// TwinCAT 3 PLC project PLCProject
// ProgramVersion: 3.1.4024.0
// libraries:
//   Tc2_MC2, * (Beckhoff Automation GmbH)
//   Tc2_MC2_Drive, * (Beckhoff Automation GmbH)
//   Tc2_NC, * (Beckhoff Automation GmbH)
//   Tc2_Standard, * (Beckhoff Automation GmbH)
//   Tc2_System, * (Beckhoff Automation GmbH)
//   Tc2_Utilities, * (Beckhoff Automation GmbH)
//   Tc3_EventLogger, * (Beckhoff Automation GmbH)
//   Tc3_Module, * (Beckhoff Automation GmbH)
// project tree:
//   DUTs/Coil Shapes/ pancake_params_0.TcDUT, racetrack_params_1.TcDUT
//   DUTs/HMI Datagrids/Inputs/ general_input_datagrid_params.TcDUT, misc_settings_input_datagrid_params.TcDUT (not stored), payoff_input_datagrid_params.TcDUT, pickup_input_datagrid_params.TcDUT
//   DUTs/HMI Datagrids/Outputs/ motor_info_datagrid.TcDUT, motor_state_datagrid.TcDUT (not stored), output_error_datagrid.TcDUT, overview_outputs_datagrid.TcDUT (not stored), payoff_output_datagrid_params.TcDUT, pickup_output_datagrid_params.TcDUT (not stored), turncount_output_datagrid.TcDUT
//   DUTs/Input Bounds/ input_bounds.TcDUT
//   DUTs/ tape_info.TcDUT
//   GVLs/ GVL.TcGVL
//   / PlcTask.TcTTO, RecipeManager.TcRMO (not stored)
//   POUs/ FB_Axis.TcPOU, FB_EventLogger.TcPOU, FB_fileReadWrite.TcPOU, FB_hmi_connection.TcPOU, FB_WindingControl.TcPOU, MAIN.TcPOU
// real-time tasks:
//   TASK PlcTask: cycle T#10ms, priority 20, ADS port 350
// motion (NC):
//   TASK NC-Task 1 SAF: cycle T#2ms, priority 4, ADS port 501
//   TASK NC-Task 1 SVB: cycle T#10ms, priority 8, ADS port 511
//   AXIS Pickup (id 1)
//     General: UnitName=°
//     Dynamic: Acceleration=2990.4, Deceleration=2990.4, Jerk=8971.19
//     Velo: RefSearch=19.93598, RefSync=19.93598, SlowManual=99.6799, FastManual=598.0794, Fast=1993.598, Maximum=1993.598
//     OtherSettings: AllowMotionCmdToSlave=true
//     encoder EncType=8
//       EncPara: ScaleFactorNumerator=360, ScaleFactorDenominator=10485760, MaxCount=#xffffffff
//     drive DrvType=9
//       DrvPara: MaxCount=#xffffffff, DriveControlDWord=#x00030100
//         Analog: VeloReferenz=2192.9578, VeloScale=1.02400649589962, TorqueSetpointScale=10, ScaleFactorActTorque=0.1
//         TimeComp: TaskDelayCycles=1
//     controller CtrType=1
//       CtrPara: PriorControlFactor=1
//         Observer: BandWidth=20
//   AXIS Payoff 1 (id 2)
//     General: UnitName=°
//     Dynamic: Acceleration=805.38, Deceleration=805.38, Jerk=2416.14
//     Velo: RefSearch=5.3692, RefSync=5.3692, SlowManual=26.846, FastManual=161.076, Fast=536.92, Maximum=536.92
//     OtherSettings: AllowMotionCmdToSlave=true
//     encoder EncType=19
//       EncPara: ScaleFactorNumerator=360, ScaleFactorDenominator=62914560, MaxCount=#xffffffff
//     drive DrvType=16
//       DrvPara: MaxCount=#xffffffff, DriveControlDWord=#x00020100
//         Analog: VeloReferenz=590.612, VeloScale=32, TorqueSetpointScale=10, ScaleFactorActTorque=0.1
//         TimeComp: TaskDelayCycles=1
//     controller CtrType=1
//       CtrPara: PriorControlFactor=1
//         Observer: BandWidth=20
//   AXIS Payoff 2 (id 3)
//     General: UnitName=°
//     Dynamic: Acceleration=805.38, Deceleration=805.38, Jerk=2416.14
//     Velo: RefSearch=5.3692, RefSync=5.3692, SlowManual=26.846, FastManual=161.076, Fast=536.92, Maximum=536.92
//     OtherSettings: AllowMotionCmdToSlave=true
//     encoder EncType=19
//       EncPara: ScaleFactorNumerator=360, ScaleFactorDenominator=62914560, MaxCount=#xffffffff
//     drive DrvType=16
//       DrvPara: MaxCount=#xffffffff, DriveControlDWord=#x00020100
//         Analog: VeloReferenz=590.612, VeloScale=32, TorqueSetpointScale=10, ScaleFactorActTorque=0.1
//         TimeComp: TaskDelayCycles=1
//     controller CtrType=1
//       CtrPara: PriorControlFactor=1
//         Observer: BandWidth=20
//   AXIS Payoff 3 (id 4)
//     General: UnitName=°
//     Dynamic: Acceleration=805.38, Deceleration=805.38, Jerk=2416.14
//     Velo: RefSearch=5.3692, RefSync=5.3692, SlowManual=26.846, FastManual=161.076, Fast=536.92, Maximum=536.92
//     OtherSettings: AllowMotionCmdToSlave=true
//     encoder EncType=19
//       EncPara: ScaleFactorNumerator=360, ScaleFactorDenominator=62914560, MaxCount=#xffffffff
//     drive DrvType=16
//       DrvPara: MaxCount=#xffffffff, DriveControlDWord=#x00020100
//         Analog: VeloReferenz=590.612, VeloScale=32, TorqueSetpointScale=10, ScaleFactorActTorque=0.1
//         TimeComp: TaskDelayCycles=1
//     controller CtrType=1
//       CtrPara: PriorControlFactor=1
//         Observer: BandWidth=20
// I/O:
//   DEVICE Device 1 (EtherCAT), AmsNetId 5.143.168.64.2.1
//     Term 9 (EK1200) [EK1200-5000 EtherCAT Power supply (2A E-Bus)]
//       Term 2 (EL3002) [EL3002 2Ch. Ana. Input +/-10V]
//       Term 3 (EL1859) [EL1859 8Ch. Dig. Input 24V, 3ms, 8Ch. Dig. Output 24V, 0.5A]
//       Term 4 (EL6070-0033) [EL6070-0033 1Ch. Licence key terminal, individual licences]
//       Term 11 (ELM7222-0011) [ELM7222-0011 2Ch. Servo Terminal (DS402, 48 V, 8 A RMS, OCT)]
//         startup 8195:21 := 0E01 // Motor Settings Ch.1 / Commutation offset
//         startup 24704:0 := 10270000 // Max motor speed Ch.1
//         startup 8196:19 := 0000 // Brake Settings Ch.1 / Emergency application timeout
//         startup 8194:51 := 0A00 // Amplifier Settings Ch.1 / Stand still window
//         startup 8194:19 := 7600 // Amplifier Settings Ch.1 / Current loop proportional gain
//         startup 8194:18 := 1300 // Amplifier Settings Ch.1 / Current loop integral time
//         startup 8194:21 := 24010000 // Amplifier Settings Ch.1 / Velocity loop proportional gain
//         startup 8194:20 := 96000000 // Amplifier Settings Ch.1 / Velocity loop integral time
//       Term 12 (ELM7222-0011) [ELM7222-0011 2Ch. Servo Terminal (DS402, 48 V, 8 A RMS, OCT)]
//         startup 8195:21 := 0E01 // Motor Settings Ch.1 / Commutation offset
//         startup 24704:0 := 10270000 // Max motor speed Ch.1
//         startup 8196:19 := 0000 // Brake Settings Ch.1 / Emergency application timeout
//         startup 8194:51 := 0A00 // Amplifier Settings Ch.1 / Stand still window
//         startup 8194:19 := 7600 // Amplifier Settings Ch.1 / Current loop proportional gain
//         startup 8194:18 := 1300 // Amplifier Settings Ch.1 / Current loop integral time
//         startup 8194:21 := 24010000 // Amplifier Settings Ch.1 / Velocity loop proportional gain
//         startup 8194:20 := 96000000 // Amplifier Settings Ch.1 / Velocity loop integral time
//         startup 10243:21 := 0E01 // Motor Settings Ch.2 / Commutation offset
//         startup 26752:0 := 10270000 // Max motor speed Ch.2
//         startup 10244:19 := 0000 // Brake Settings Ch.2 / Emergency application timeout
//         startup 10242:51 := 0A00 // Amplifier Settings Ch.2 / Stand still window
//         startup 10242:19 := 7600 // Amplifier Settings Ch.2 / Current loop proportional gain
//         startup 10242:18 := 1300 // Amplifier Settings Ch.2 / Current loop integral time
//         startup 10242:21 := 24010000 // Amplifier Settings Ch.2 / Velocity loop proportional gain
//         startup 10242:20 := 96000000 // Amplifier Settings Ch.2 / Velocity loop integral time
//       Term 13 (EK1110) [EK1110 EtherCAT extension]
//     Drive 16 (AX5103-0000-0214) [AX5103-0000-0214 EtherCAT Drive (SoE, 1 Ch.)]
// variable links:
//   NC-Task 1 SAF/Axes/Payoff 1 <-> Device 1 (EtherCAT)/Term 9 (EK1200)/Term 12 (ELM7222-0011)
//     Drive/Inputs/In/nDataIn1 <-> DS402 Following error actual value Channel 2/Following error actual value
//     Drive/Inputs/In/nDataIn3[0] <-> DS402 Torque actual value Channel 2/Torque actual value
//     Drive/Inputs/In/nDcOutputTime <-> InfoData/DcOutputShift
//     Drive/Inputs/In/nState1 <-> DS402 Statusword Channel 2/Statusword
//     Drive/Inputs/In/nState2 <-> DS402 Statusword Channel 2/Statusword @bit 8
//     Drive/Inputs/In/nState4 @bit 1 <-> WcState/InputToggle
//     Drive/Inputs/In/nState4 <-> WcState/WcState
//     Drive/Inputs/In/nState5 <-> DS402 Modes of operation display Channel 2/Modes of operation display
//     Drive/Outputs/Out/nCtrl1 <-> DS402 Controlword Channel 2/Controlword
//     Drive/Outputs/Out/nCtrl2 <-> DS402 Controlword Channel 2/Controlword @bit 8
//     Drive/Outputs/Out/nCtrl5 <-> DS402 Modes of operation Channel 2/Modes of operation
//     Drive/Outputs/Out/nDataOut1 <-> DS402 Target position Channel 2/Target position
//     Drive/Outputs/Out/nDataOut4[0] <-> DS402 Target torque Channel 2/Target torque
//     Drive/Outputs/Out/nDataOut5 <-> DS402 High velocity limit value Channel 2/High velocity limit value
//     Drive/Outputs/Out/nDataOut6 <-> DS402 Low velocity limit value Channel 2/Low velocity limit value
//     Enc/Inputs/In/nDataIn1 <-> DS402 Position actual value Channel 2/Position actual value
//     Enc/Inputs/In/nDcInputTime <-> InfoData/DcInputShift
//     Enc/Inputs/In/nState4 @bit 1 <-> WcState/InputToggle
//     Enc/Inputs/In/nState4 <-> WcState/WcState
//   NC-Task 1 SAF/Axes/Payoff 2 <-> Device 1 (EtherCAT)/Term 9 (EK1200)/Term 11 (ELM7222-0011)
//     Drive/Inputs/In/nDataIn1 <-> DS402 Following error actual value Channel 1/Following error actual value
//     Drive/Inputs/In/nDataIn3[0] <-> DS402 Torque actual value Channel 1/Torque actual value
//     Drive/Inputs/In/nDcOutputTime <-> InfoData/DcOutputShift
//     Drive/Inputs/In/nState1 <-> DS402 Statusword Channel 1/Statusword
//     Drive/Inputs/In/nState2 <-> DS402 Statusword Channel 1/Statusword @bit 8
//     Drive/Inputs/In/nState4 @bit 1 <-> WcState/InputToggle
//     Drive/Inputs/In/nState4 <-> WcState/WcState
//     Drive/Inputs/In/nState5 <-> DS402 Modes of operation display Channel 1/Modes of operation display
//     Drive/Outputs/Out/nCtrl1 <-> DS402 Controlword Channel 1/Controlword
//     Drive/Outputs/Out/nCtrl2 <-> DS402 Controlword Channel 1/Controlword @bit 8
//     Drive/Outputs/Out/nCtrl5 <-> DS402 Modes of operation Channel 1/Modes of operation
//     Drive/Outputs/Out/nDataOut1 <-> DS402 Target position Channel 1/Target position
//     Drive/Outputs/Out/nDataOut4[0] <-> DS402 Target torque Channel 1/Target torque
//     Drive/Outputs/Out/nDataOut5 <-> DS402 High velocity limit value Channel 1/High velocity limit value
//     Drive/Outputs/Out/nDataOut6 <-> DS402 Low velocity limit value Channel 1/Low velocity limit value
//     Enc/Inputs/In/nDataIn1 <-> DS402 Position actual value Channel 1/Position actual value
//     Enc/Inputs/In/nDcInputTime <-> InfoData/DcInputShift
//     Enc/Inputs/In/nState4 @bit 1 <-> WcState/InputToggle
//     Enc/Inputs/In/nState4 <-> WcState/WcState
//   NC-Task 1 SAF/Axes/Payoff 3 <-> Device 1 (EtherCAT)/Term 9 (EK1200)/Term 12 (ELM7222-0011)
//     Drive/Inputs/In/nDataIn1 <-> DS402 Following error actual value Channel 1/Following error actual value
//     Drive/Inputs/In/nDataIn3[0] <-> DS402 Torque actual value Channel 1/Torque actual value
//     Drive/Inputs/In/nDcOutputTime <-> InfoData/DcOutputShift
//     Drive/Inputs/In/nState1 <-> DS402 Statusword Channel 1/Statusword
//     Drive/Inputs/In/nState2 <-> DS402 Statusword Channel 1/Statusword @bit 8
//     Drive/Inputs/In/nState4 @bit 1 <-> WcState/InputToggle
//     Drive/Inputs/In/nState4 <-> WcState/WcState
//     Drive/Inputs/In/nState5 <-> DS402 Modes of operation display Channel 1/Modes of operation display
//     Drive/Outputs/Out/nCtrl1 <-> DS402 Controlword Channel 1/Controlword
//     Drive/Outputs/Out/nCtrl2 <-> DS402 Controlword Channel 1/Controlword @bit 8
//     Drive/Outputs/Out/nCtrl5 <-> DS402 Modes of operation Channel 1/Modes of operation
//     Drive/Outputs/Out/nDataOut1 <-> DS402 Target position Channel 1/Target position
//     Drive/Outputs/Out/nDataOut4[0] <-> DS402 Target torque Channel 1/Target torque
//     Drive/Outputs/Out/nDataOut5 <-> DS402 High velocity limit value Channel 1/High velocity limit value
//     Drive/Outputs/Out/nDataOut6 <-> DS402 Low velocity limit value Channel 1/Low velocity limit value
//     Enc/Inputs/In/nDataIn1 <-> DS402 Position actual value Channel 1/Position actual value
//     Enc/Inputs/In/nDcInputTime <-> InfoData/DcInputShift
//     Enc/Inputs/In/nState4 @bit 1 <-> WcState/InputToggle
//     Enc/Inputs/In/nState4 <-> WcState/WcState
//   NC-Task 1 SAF/Axes/Pickup <-> Device 1 (EtherCAT)/Drive 16 (AX5103-0000-0214)
//     Drive/Inputs/In/nDataIn1 <-> AT/Following distance
//     Drive/Inputs/In/nDataIn3[0] <-> AT/Torque/force feedback value
//     Drive/Inputs/In/nDcOutputTime <-> InfoData/DcOutputShift
//     Drive/Inputs/In/nState1 <-> AT/Drive status word @bit 8
//     Drive/Inputs/In/nState2 <-> AT/Drive status word
//     Drive/Inputs/In/nState4 @bit 1 <-> WcState/InputToggle
//     Drive/Inputs/In/nState4 <-> WcState/WcState
//     Drive/Outputs/Out/nCtrl1 <-> MDT/Master control word @bit 8
//     Drive/Outputs/Out/nDataOut1 <-> MDT/Position command value
//     Drive/Outputs/Out/nDataOut4[0] <-> MDT/Torque/force command value
//     Drive/Outputs/Out/nDataOut5 <-> MDT/High velocity limit value
//     Drive/Outputs/Out/nDataOut6 <-> MDT/Low velocity limit value
//     Enc/Inputs/In/nDataIn1 <-> AT/Position feedback 1 value
//     Enc/Inputs/In/nDcInputTime <-> InfoData/DcInputShift
//     Enc/Inputs/In/nState4 @bit 1 <-> WcState/InputToggle
//     Enc/Inputs/In/nState4 <-> WcState/WcState
//   PLCProject/PLCProject Instance <-> NC-Task 1 SAF/Axes/Payoff 1
//     PlcTask Inputs/MAIN.FB_WindingControl.payoff_axis_list[1].AXIS.NcToPlc <-> Outputs/ToPlc
//     PlcTask Outputs/MAIN.FB_WindingControl.payoff_axis_list[1].AXIS.PlcToNc <-> Inputs/FromPlc
//   PLCProject/PLCProject Instance <-> NC-Task 1 SAF/Axes/Payoff 2
//     PlcTask Inputs/MAIN.FB_WindingControl.payoff_axis_list[2].AXIS.NcToPlc <-> Outputs/ToPlc
//     PlcTask Outputs/MAIN.FB_WindingControl.payoff_axis_list[2].AXIS.PlcToNc <-> Inputs/FromPlc
//   PLCProject/PLCProject Instance <-> NC-Task 1 SAF/Axes/Payoff 3
//     PlcTask Inputs/MAIN.FB_WindingControl.payoff_axis_list[3].AXIS.NcToPlc <-> Outputs/ToPlc
//     PlcTask Outputs/MAIN.FB_WindingControl.payoff_axis_list[3].AXIS.PlcToNc <-> Inputs/FromPlc
//   PLCProject/PLCProject Instance <-> NC-Task 1 SAF/Axes/Pickup
//     PlcTask Inputs/MAIN.FB_WindingControl.pickup_axis_list[1].AXIS.NcToPlc <-> Outputs/ToPlc
//     PlcTask Outputs/MAIN.FB_WindingControl.pickup_axis_list[1].AXIS.PlcToNc <-> Inputs/FromPlc

CONFIGURATION PLCProject
    RESOURCE PLC ON TwinCAT3
        TASK PlcTask(INTERVAL := T#10ms, PRIORITY := 20);
        PROGRAM MAIN WITH PlcTask : MAIN;
    END_RESOURCE
END_CONFIGURATION

// ---- DUTs/Coil Shapes/pancake_params_0.TcDUT
TYPE pancake_params_0 :
STRUCT
	radius : LREAL := 200; // radius of pancake coil in mm
END_STRUCT
END_TYPE

// ---- DUTs/Coil Shapes/racetrack_params_1.TcDUT
//Defining our dimensions for our racetrack coil
TYPE racetrack_params_1 :
STRUCT
	length : LREAL := 150; //mm
	radius : LREAL := 100; //mm
END_STRUCT
END_TYPE

// ---- DUTs/HMI Datagrids/Inputs/general_input_datagrid_params.TcDUT
TYPE general_input_datagrid_params :
STRUCT
	tension : LREAL :=10;
	linspeed : LREAL:=0.5;
	unwinding : BOOL;
END_STRUCT
END_TYPE

// ---- DUTs/HMI Datagrids/Inputs/payoff_input_datagrid_params.TcDUT
TYPE payoff_input_datagrid_params :
STRUCT
	motor_name : STRING;
	tape_type : INT :=1;
	coil_type : INT :=1;
	radius : LREAL :=150;
	enabled : BOOL ;
END_STRUCT
END_TYPE

// ---- DUTs/HMI Datagrids/Inputs/pickup_input_datagrid_params.TcDUT
TYPE pickup_input_datagrid_params :
STRUCT
	motor_name : STRING;
	turn_count: INT :=1;
	coil_shape: INT :=0;
END_STRUCT
END_TYPE

// ---- DUTs/HMI Datagrids/Outputs/motor_info_datagrid.TcDUT
TYPE motor_info_datagrid :
STRUCT
	speed : LREAL;
	torque : LREAL;
	errortype : UDINT;
	errorid : UDINT;
	currentRadius: LREAL;
END_STRUCT
END_TYPE

// ---- DUTs/HMI Datagrids/Outputs/output_error_datagrid.TcDUT
TYPE output_error_datagrid :
STRUCT
	errorStatus : BOOL;
	errorID : UDINT;
END_STRUCT
END_TYPE

// ---- DUTs/HMI Datagrids/Outputs/payoff_output_datagrid_params.TcDUT
TYPE payoff_output_datagrid_params :
STRUCT
	motor_name: STRING;
	rpm : LREAL;
	linear_speed : LREAL;
	turn_count : LREAL;
	enabled : BOOL ;
END_STRUCT
END_TYPE

// ---- DUTs/HMI Datagrids/Outputs/turncount_output_datagrid.TcDUT
TYPE turncount_output_datagrid :
STRUCT
	
	pickupTC1 : LREAL;
	payoffTC1 : LREAL;
	payoffTC2 : LREAL;
	payoffTC3 : LREAL;
END_STRUCT
END_TYPE

// ---- DUTs/Input Bounds/input_bounds.TcDUT
//defines bounds for all HMI inputs
TYPE input_bounds :
STRUCT
	
	linear_speed_low : LREAL := 0.01; //(m/s)
	linear_speed_high: LREAL := 1.0;  //(m/s)

	tension_low : LREAL := 5; //(N)
	tension_high : LREAL := 20; //(N)
	
	turn_count_pickup_low : INT := 1;
	turn_count_pickup_high : INT := 1000;
	
	radius_payoff_low : LREAL:=GVL.MIN_MOUNT_RADIUS; //(mm)
	radius_payoff_high : LREAL:=GVL.MAX_PAYOFF_RADIUS-10; //(mm)
	
	radius_pickup_pancake_low : LREAL:=GVL.MIN_MOUNT_RADIUS; //((mm)
	radius_pickup_pancake_high: LREAL:=GVL.MAX_PICKUP_RADIUS-10; //(mm)
	
	coil_shape_low : INT :=0;
	coil_shape_high : INT :=2;
	
	acceleration_low : LREAL :=0.1; //(m/s)
	acceleration_high : LREAL :=1; //(m/s)
	
	decceleration_low : LREAL :=0.1; //(m^2/s)
	decelleration_high : LREAL :=1; //(m^2/s)

	jerk_low : LREAL:=0.1;
	jerk_high : LREAL:=1;
	
END_STRUCT
END_TYPE

// ---- DUTs/tape_info.TcDUT
//material properties of the tape
TYPE tape_info :
STRUCT
	tape_width: LREAL:=4.0;
	tape_depth: LREAL:=0.1;
	mass_per_cm_g : LREAL :=10;
END_STRUCT
END_TYPE

// ---- GVLs/GVL.TcGVL
{attribute 'qualified_only'}
VAR_GLOBAL CONSTANT
	MAX_PAYOFF_COUNT : INT:=3;
	MAX_PICKUP_COUNT : INT:=1;
	
	MAX_CSV_ROWS : INT:=8;
	MAX_CSV_COLUMNS : INT:=1;
	MAX_CSV_FIELD_LENGTH: INT:=128;
	
	
	MIN_MOUNT_RADIUS: LREAL := 113; //(mm)
	
	//found from hardware. specific to each type of motor
	PICKUP_RATED_CURRENT : LREAL :=11.8;
	PICKUP_TORQUE_CONSTANT: LREAL :=1.9;
	PAYOFF_RATED_CURRENT: LREAL :=8;
	PAYOFF_TORQUE_CONSTANT: LREAL :=0.1;
	
	TAPE1_WIDTH: LREAL :=4.0;
	TAPE1_DEPTH: LREAL := 0.1;
	TAPE1_MASS_PER_CM_G : LREAL :=10;
	
	TAPE2_WIDTH: LREAL :=4.0;
	TAPE2_DEPTH: LREAL := 0.1;
	TAPE2_MASS_PER_CM_G : LREAL :=10;
	
	//LIMITS
	
	INNER_RADIUS : LREAL:= 133; //(mm)
	
	MAX_PICKUP_RADIUS : LREAL:=250;
	MAX_PAYOFF_RADIUS : LREAL:=200;
	
	MIN_THRESHOLD_TORQUE : LREAL:= 2;
	
	MAX_EVENT_SIZE : INT:= 50;
END_VAR

// ---- POUs/MAIN.TcPOU
PROGRAM MAIN
VAR
	InitComplete: BOOL;
	
	//Function Block INIT
	FB_hmi_connection: FB_hmi_connection;
	FB_WindingControl: FB_WindingControl;
	FB_EventLogger: FB_EventLogger;
	FB_FileReadWrite: FB_fileReadWrite;
	
	
	
	
END_VAR

CYCLIC();

METHOD CYCLIC : BOOL
VAR_INPUT
END_VAR
IF NOT InitComplete THEN
    InitComplete := INIT();
    RETURN;
END_IF

//FB Cyclic logic. 

FB_EventLogger.CYCLIC(); //event logger
FB_hmi_connection.CYCLIC(); //hmi inputs and outputs
FB_WindingControl.CYCLIC(); //motor control. 
FB_FileReadWrite.CYCLIC();
END_METHOD

METHOD INIT : BOOL
VAR_INPUT
END_VAR
//Function Block INIT
FB_hmi_connection.INIT();
FB_WindingControl.INIT();
FB_EventLogger.INIT();
//MAIN INIT


FB_WindingControl.hmiConnection:=ADR(FB_hmi_connection);
FB_WindingControl.eventLogger:=ADR(FB_EventLogger);
FB_WindingControl.fileReadWrite:=ADR(FB_fileReadWrite);

INIT:=TRUE;
END_METHOD

END_PROGRAM

// ---- POUs/FB_hmi_connection.TcPOU
FUNCTION_BLOCK FB_hmi_connection
VAR_INPUT
    // Datagrid parameters
    payoff_input_datagrid_params_list        : ARRAY[1..GVL.MAX_PAYOFF_COUNT] OF payoff_input_datagrid_params;
    payoff_output_datagrid_params_list       : ARRAY[1..GVL.MAX_PAYOFF_COUNT] OF payoff_output_datagrid_params;
    pickup_input_datagrid_params_list        : ARRAY[1..GVL.MAX_PICKUP_COUNT] OF pickup_input_datagrid_params;
    pickup_output_datagrid_params_list       : ARRAY[1..GVL.MAX_PICKUP_COUNT] OF pickup_output_datagrid_params;
    general_input_datagrid_params_list       : ARRAY[1..1] OF general_input_datagrid_params;
    misc_settings_input_datagrid_params_list : ARRAY[1..1] OF misc_settings_input_datagrid_params;
    pickup_pancake_input_datagrid_params_list: ARRAY[1..1] OF pancake_params_0;
    pickup_racetrack_input_datagrid_params_list: ARRAY[1..1] OF racetrack_params_1;
    output_error_datagrid_list               : ARRAY[0..3] OF output_error_datagrid;
    motor_state_datagrid_list                : ARRAY[0..3] OF motor_state_datagrid;
    overview_outputs_datagrid_list           : ARRAY[1..1] OF overview_outputs_datagrid;
    turncount_output_datagrid_list           : ARRAY[1..1] OF turncount_output_datagrid;
    motor_info_datagrid_list                 : ARRAY[1..4] OF motor_info_datagrid;
    color_list                               : ARRAY[0..3] OF DWORD;

    // Outputs
    motor_turncount                          : ARRAY[1..4] OF DINT;
    userNote                                 : STRING := '';

    // Hardware inputs
    estopHW AT %I*                           : BOOL := FALSE;

    // Control page
    resetUI                                  : BOOL;
    startUI                                  : BOOL;
    tensionUI                                : BOOL;
    homeUI                                   : BOOL;
    freespinUI                               : BOOL;
    clearUI                                  : BOOL;
	
    // Historized variables
    torque                                   : ARRAY[1..GVL.MAX_PAYOFF_COUNT+GVL.MAX_PICKUP_COUNT] OF LREAL;
    rpm                                      : ARRAY[1..GVL.MAX_PAYOFF_COUNT+GVL.MAX_PICKUP_COUNT] OF LREAL;

    // Misc
    state                                    : INT := 0;

    // User ID
    user                                     : STRING(255) := 'N/A';
END_VAR

METHOD CYCLIC : BOOL
VAR_INPUT
END_VAR

VAR

END_VAR
END_METHOD

METHOD INIT : BOOL
VAR_INPUT
END_VAR
init_datagrids();
END_METHOD

METHOD init_datagrids : BOOL
VAR_INPUT
END_VAR

VAR
	i: INT;
END_VAR
//initalize datagrids for ui
FOR i := 1 TO GVL.MAX_PAYOFF_COUNT DO
	
	payoff_input_datagrid_params_list[i].motor_name := TO_STRING(i);
	payoff_output_datagrid_params_list[i].motor_name := TO_STRING(i);
		
END_FOR;

pickup_input_datagrid_params_list[1].motor_name := TO_STRING(1);
pickup_output_datagrid_params_list[1].motor_name := TO_STRING(1);
END_METHOD

END_FUNCTION_BLOCK

// ---- POUs/FB_WindingControl.TcPOU
FUNCTION_BLOCK FB_WindingControl
VAR_INPUT
	// Input hmi connection from MAIN
	hmiConnection   : POINTER TO FB_hmi_connection;   // HMI connection
	eventLogger     : POINTER TO FB_EventLogger;      // Event logger
	fileReadWrite   : POINTER TO FB_fileReadWrite;    // File read/write
END_VAR

VAR
	// Temporary testing vars
	dist : LREAL ;
	testing : BOOL;
	// Function Blocks

	// CONTROL VARS
	desiredTension          : LREAL := 0;         // Desired tension
	desiredLinspeed         : LREAL := 0;         // Desired linear speed
	unwinding               : BOOL  := FALSE;     // Unwinding flag
	desiredTurnCountPickup  : DINT  := 0;         // Desired turn count for pickup
	
	// Exit conditions
	target_turn_count       : DINT  := 0;         // Target turn count post gear ratio

	// STATUS VARS
	state                   : INT   := 0;         // State for state machine
	cnt                     : UINT  := 0;         // PLC cycle counter
	eta                     : LREAL := 0;         // Time till completion in seconds
	etaFormattedString      : STRING(255);        // Formatted ETA in format ETA: M:S
	progressPercent         : LREAL := 0;         // Progress percentage (0 to 100) based on turn count

	actualLinspeed			: LREAL := 0;
	// COIL MODELS (currently not used)
	// coil_model_base_Xcords : ARRAY[0..MAX_COIL_TYPE_COUNT] OF ARRAY[1..MAX_SIZE_COIL_MODEL] OF LREAL;
	// coil_model_base_Ycords : ARRAY[0..MAX_COIL_TYPE_COUNT] OF ARRAY[1..MAX_SIZE_COIL_MODEL] OF LREAL;

	// coil_model_rot_Xcords  : ARRAY[0..MAX_COIL_TYPE_COUNT] OF ARRAY[1..MAX_SIZE_COIL_MODEL] OF LREAL;
	// coil_model_rot_Ycords  : ARRAY[0..MAX_COIL_TYPE_COUNT] OF ARRAY[1..MAX_SIZE_COIL_MODEL] OF LREAL;

	// AXIS LIST
	payoff_axis_list        : ARRAY[1..GVL.MAX_PAYOFF_COUNT] OF FB_Axis;   // Payoff axis list
	pickup_axis_list        : ARRAY[1..GVL.MAX_PICKUP_COUNT] OF FB_Axis;   // Pickup axis list
	axis_list 				: ARRAY[1..GVL.MAX_PAYOFF_COUNT+GVL.MAX_PICKUP_COUNT] OF POINTER TO FB_Axis; //contains pointers to all axies. 1 being pickup, 2,3,4 being payoff
	// MISC
	tape_info 				: ARRAY[0..10] OF tape_info;
	numOfEnabledPayoff      : INT := 0;           // Number of enabled payoffs
	tStart                  : TIME;               // Start time
	tEnd                    : TIME;               // End time
	tElapsed                : TIME;               // Elapsed time
	allowInputEdits 		: BOOL;				  //enables/disable input mods


END_VAR

VAR CONSTANT
	input_bounds            : input_bounds;       // Input bounds
	MAX_COIL_TYPE_COUNT     : INT := 1;           // Number of coil types (counts from 0)
	MAX_SIZE_COIL_MODEL     : INT := 1205;        // Maximum size of coil model
	TARGET_PICKUP_FORCE     : LREAL := 10;        // Target pickup force
	pi                      : LREAL := 4 * ATAN(1); // PI for math reasons (might be built-in but couldn't find it)
END_VAR

METHOD accelerating_tension : BOOL
VAR_INPUT
END_VAR

VAR
	i: INT;
	pickupLinspeed: LREAL;
	dist: LREAL;
	desiredVelocity: LREAL;
	adjustedVelocity: LREAL;
END_VAR
winding_tension();
END_METHOD

METHOD all_check : BOOL
VAR_INPUT
	write: BOOL;
END_VAR
all_check:= all_check OR general_input_check(write:=write);
all_check:= all_check OR payoff_input_check(write:=write);
all_check:=all_check OR pickup_input_check(write:=write);
END_METHOD

METHOD count_enabled_motors : BOOL
VAR_INPUT
END_VAR

VAR
	i: INT;
END_VAR
 //updates status of all axises, pickup and payoff

numOfEnabledPayoff:=0;

FOR i:= 1 TO GVL.MAX_PAYOFF_COUNT DO
IF	payoff_axis_list[i].enabled THEN
	numOfEnabledPayoff:=numOfEnabledPayoff+1;
END_IF
END_FOR
END_METHOD

METHOD CYCLIC : BOOL
VAR
	
	i: INT;
	

	intital: BOOL;
	errorOutput: BOOL;
	errorStatus: BOOL;
	
END_VAR
//cycle counter
cnt := cnt +1;

//-------------------------------------------------------------------------------------------------------------- USER INPUT --------------------------------------------------------------------------------------------------------------
CASE state OF
    10:
    // ========================================10========================================
    IF hmiConnection^.resetUI THEN
        reset();
        hmiConnection^.resetUI := FALSE;
    END_IF

    IF hmiConnection^.startUI THEN
        ADSLOGSTR(msgCtrlMask := ADSLOG_MSGTYPE_ERROR OR ADSLOG_MSGTYPE_MSGBOX,
                  msgFmtStr := 'Error Occured. Unable to start winding while not in tension state',
                  strArg := '');
        hmiConnection^.startUI := FALSE;
    END_IF

    IF hmiConnection^.tensionUI THEN
        state := 20;
        errorOutput := TRUE;
    END_IF

    transfer_hmi_vars();

    IF hmiConnection^.homeUI THEN
        state := 50;
        errorOutput := TRUE;
    END_IF

    IF hmiConnection^.estopHW THEN
        state := 500;
    END_IF

    IF hmiConnection^.freespinUI THEN
        state := 11;
    END_IF

    // ========================================10========================================

    11:
    // ========================================11========================================
    IF NOT hmiConnection^.freespinUI THEN
        state := 10;
    END_IF

    IF hmiConnection^.resetUI THEN
        reset();
        hmiConnection^.resetUI := FALSE;
    END_IF

    IF hmiConnection^.startUI THEN
        ADSLOGSTR(msgCtrlMask := ADSLOG_MSGTYPE_ERROR OR ADSLOG_MSGTYPE_MSGBOX,
                  msgFmtStr := 'Error Occured. Unable to start winding while not in tension state',
                  strArg := '');
        hmiConnection^.startUI := FALSE;
    END_IF

    IF hmiConnection^.tensionUI THEN
        ADSLOGSTR(msgCtrlMask := ADSLOG_MSGTYPE_ERROR OR ADSLOG_MSGTYPE_MSGBOX,
                  msgFmtStr := 'Error Occured. Unable to start tension while in freespin state',
                  strArg := '');
        hmiConnection^.tensionUI := FALSE;
    END_IF

    IF hmiConnection^.homeUI THEN
        state := 50;
        errorOutput := TRUE;
    END_IF

    IF hmiConnection^.estopHW THEN
        state := 500;
    END_IF

    transfer_hmi_vars();
    // ========================================11========================================

    20, 21:
    // ========================================20========================================
    IF hmiConnection^.freespinUI THEN
        ADSLOGSTR(msgCtrlMask := ADSLOG_MSGTYPE_ERROR OR ADSLOG_MSGTYPE_MSGBOX,
                  msgFmtStr := 'Error Occured. Unable to start freespin while not in standby state',
                  strArg := '');
        hmiConnection^.freespinUI := FALSE;
    END_IF

    IF hmiConnection^.resetUI THEN
        reset();
        hmiConnection^.resetUI := FALSE;
    END_IF

    IF hmiConnection^.startUI THEN
        state := 30;
        errorOutput := TRUE;
    END_IF

    IF NOT hmiConnection^.tensionUI THEN
        state := 10;
        errorOutput := TRUE;
    END_IF

    transfer_hmi_vars();

    IF hmiConnection^.homeUI THEN
        ADSLOGSTR(msgCtrlMask := ADSLOG_MSGTYPE_ERROR OR ADSLOG_MSGTYPE_MSGBOX,
                  msgFmtStr := 'Error Occured. Unable to home outside of standby state',
                  strArg := '');
        hmiConnection^.homeUI := FALSE;
    END_IF

    IF hmiConnection^.estopHW THEN
        state := 500;
    END_IF
    // ========================================20========================================

    30, 31, 32, 33:
    // ========================================30========================================
    IF hmiConnection^.freespinUI THEN
        ADSLOGSTR(msgCtrlMask := ADSLOG_MSGTYPE_ERROR OR ADSLOG_MSGTYPE_MSGBOX,
                  msgFmtStr := 'Error Occured. Unable to start freespin while not in standby state',
                  strArg := '');
        hmiConnection^.freespinUI := FALSE;
    END_IF

    IF hmiConnection^.resetUI THEN
        ADSLOGSTR(msgCtrlMask := ADSLOG_MSGTYPE_ERROR OR ADSLOG_MSGTYPE_MSGBOX,
                  msgFmtStr := 'Error Occured. Unable to reset during winding. Please pause winding.',
                  strArg := '');
        hmiConnection^.resetUI := FALSE;
    END_IF

    IF NOT hmiConnection^.startUI THEN
        state := 20;
        errorOutput := TRUE;
    END_IF

    IF NOT hmiConnection^.tensionUI THEN
        hmiConnection^.startUI := FALSE;
        state := 10;
        errorOutput := TRUE;
    END_IF

    IF hmiConnection^.checkInputsUI THEN
        all_check(write := FALSE);
        hmiConnection^.checkInputsUI := FALSE;
        errorOutput := TRUE;
    END_IF

    IF hmiConnection^.updateInputsUI THEN
        all_check(write := TRUE);
        hmiConnection^.updateInputsUI := FALSE;
    END_IF

    IF hmiConnection^.homeUI THEN
        ADSLOGSTR(msgCtrlMask := ADSLOG_MSGTYPE_ERROR OR ADSLOG_MSGTYPE_MSGBOX,
                  msgFmtStr := 'Error Occured. Unable to home outside of standby state',
                  strArg := '');
        hmiConnection^.homeUI := FALSE;
    END_IF

    IF hmiConnection^.estopHW THEN
        state := 500;
    END_IF
    // ========================================30========================================

    40, 41:
    // ========================================40========================================
    IF hmiConnection^.freespinUI THEN
        ADSLOGSTR(msgCtrlMask := ADSLOG_MSGTYPE_ERROR OR ADSLOG_MSGTYPE_MSGBOX,
                  msgFmtStr := 'Error Occured. Unable to start freespin while not in standby state',
                  strArg := '');
        hmiConnection^.freespinUI := FALSE;
    END_IF

    IF hmiConnection^.tensionUI THEN
        state := 40;
        errorOutput := TRUE;
    ELSE
        state := 41;
    END_IF

    IF hmiConnection^.resetUI THEN
        reset();
        hmiConnection^.resetUI := FALSE;
    END_IF

    IF hmiConnection^.startUI THEN
        ADSLOGSTR(msgCtrlMask := ADSLOG_MSGTYPE_ERROR OR ADSLOG_MSGTYPE_MSGBOX,
                  msgFmtStr := 'Error Occured. Unable to start while finished. Please reset first.',
                  strArg := '');
        hmiConnection^.startUI := FALSE;
    END_IF

    IF hmiConnection^.checkInputsUI THEN
        all_check(write := FALSE);
        hmiConnection^.checkInputsUI := FALSE;
    END_IF

    IF hmiConnection^.updateInputsUI THEN
        all_check(write := TRUE);
        hmiConnection^.updateInputsUI := FALSE;
    END_IF

    IF hmiConnection^.homeUI THEN
        ADSLOGSTR(msgCtrlMask := ADSLOG_MSGTYPE_ERROR OR ADSLOG_MSGTYPE_MSGBOX,
                  msgFmtStr := 'Error Occured. Unable to home outside of standby state',
                  strArg := '');
        hmiConnection^.homeUI := FALSE;
    END_IF

    IF hmiConnection^.estopHW THEN
        state := 500;
    END_IF
    // ========================================40========================================

    400:
    // ========================================400========================================
    IF hmiConnection^.freespinUI THEN
        ADSLOGSTR(msgCtrlMask := ADSLOG_MSGTYPE_ERROR OR ADSLOG_MSGTYPE_MSGBOX,
                  msgFmtStr := 'Error Occured. Unable to start freespin while not in standby state',
                  strArg := '');
        hmiConnection^.freespinUI := FALSE;
    END_IF

    IF hmiConnection^.resetUI THEN
        reset();
        state := 10;
        hmiConnection^.resetUI := FALSE;
        errorOutput := TRUE;
    END_IF

    IF hmiConnection^.startUI THEN
        ADSLOGSTR(msgCtrlMask := ADSLOG_MSGTYPE_ERROR OR ADSLOG_MSGTYPE_MSGBOX,
                  msgFmtStr := 'Error Occured. Unable to start while in error state. Please reset first, and resolve error.',
                  strArg := '');
        hmiConnection^.resetUI := FALSE;
    END_IF

    IF hmiConnection^.checkInputsUI THEN
        all_check(write := FALSE);
        hmiConnection^.checkInputsUI := FALSE;
    END_IF

    IF hmiConnection^.updateInputsUI THEN
        all_check(write := TRUE);
        hmiConnection^.updateInputsUI := FALSE;
    END_IF

    IF hmiConnection^.homeUI THEN
        ADSLOGSTR(msgCtrlMask := ADSLOG_MSGTYPE_ERROR OR ADSLOG_MSGTYPE_MSGBOX,
                  msgFmtStr := 'Error Occured. Unable to home inside error state. Please resolve errors on enabled axises',
                  strArg := '');
        hmiConnection^.homeUI := FALSE;
    END_IF

    IF hmiConnection^.estopHW THEN
        state := 500;
    END_IF
    // ========================================400========================================

    50:
    // ========================================50========================================
    IF hmiConnection^.tensionUI THEN
        ADSLOGSTR(msgCtrlMask := ADSLOG_MSGTYPE_ERROR OR ADSLOG_MSGTYPE_MSGBOX,
                  msgFmtStr := 'Error Occured. Unable to tension while in homing sdtate. Please stop homing.',
                  strArg := '');
        hmiConnection^.resetUI := FALSE;
    END_IF

    IF hmiConnection^.resetUI THEN
        reset();
        state := 10;
        hmiConnection^.resetUI := FALSE;
        errorOutput := TRUE;
    END_IF

    IF hmiConnection^.startUI THEN
        ADSLOGSTR(msgCtrlMask := ADSLOG_MSGTYPE_ERROR OR ADSLOG_MSGTYPE_MSGBOX,
                  msgFmtStr := 'Error Occured. Unable to start while in homing sdtate. Please stop homing.',
                  strArg := '');
        hmiConnection^.resetUI := FALSE;
    END_IF

    transfer_hmi_vars();

    IF hmiConnection^.homeUI THEN
        hmiConnection^.homeUI := FALSE;
        state := 10;
        errorOutput := TRUE;
    END_IF

    IF hmiConnection^.estopHW THEN
        state := 500;
    END_IF
    // ========================================50========================================

    500:
    // ========================================500========================================
    IF hmiConnection^.tensionUI THEN
        ADSLOGSTR(msgCtrlMask := ADSLOG_MSGTYPE_ERROR OR ADSLOG_MSGTYPE_MSGBOX,
                  msgFmtStr := 'Error Occured. Unable to tension while in ESTOP state. Please reset first.',
                  strArg := '');
        hmiConnection^.tensionUI := FALSE;
    END_IF

    IF hmiConnection^.resetUI THEN
        reset();
        state := 10;
        hmiConnection^.resetUI := FALSE;
        errorOutput := TRUE;
    END_IF

    IF hmiConnection^.startUI THEN
        ADSLOGSTR(msgCtrlMask := ADSLOG_MSGTYPE_ERROR OR ADSLOG_MSGTYPE_MSGBOX,
                  msgFmtStr := 'Error Occured. Unable to start while in ESTOP state. Please reset first.',
                  strArg := '');
        hmiConnection^.startUI := FALSE;
    END_IF

    IF hmiConnection^.checkInputsUI THEN
        all_check(write := FALSE);
        hmiConnection^.checkInputsUI := FALSE;
    END_IF

    IF hmiConnection^.updateInputsUI THEN
        all_check(write := TRUE);
        hmiConnection^.updateInputsUI := FALSE;
    END_IF

    IF hmiConnection^.homeUI THEN
        ADSLOGSTR(msgCtrlMask := ADSLOG_MSGTYPE_ERROR OR ADSLOG_MSGTYPE_MSGBOX,
                  msgFmtStr := 'Error Occured. Unable to home while in ESTOP state. Please reset first.',
                  strArg := '');
        hmiConnection^.homeUI := FALSE;
    END_IF

    IF hmiConnection^.estopHW THEN
        state := 500;
    END_IF
    // ========================================500========================================
END_CASE
//-------------------------------------------------------------------------------------------------------------- USER INPUT --------------------------------------------------------------------------------------------------------------
	
//clear status vars for axis. we will update them depending on our current state.
pickup_axis_list[1].setClear();

FOR i:= 1 TO GVL.MAX_PAYOFF_COUNT DO
	payoff_axis_list[i].setClear();
END_FOR

//check FOR error, IF error THEN set state TO 400

general_error_check(errorStatus=>errorStatus,errorOutput:=errorOutput);


//if no error, but currently in error state set winding to standby
//if none of the above state is unmodified
IF errorStatus THEN
	state:=400;
ELSIF state=400 AND NOT errorStatus THEN
	state:=10;
END_IF

//update HMI with certain motor values. 
hmi_update();
find_actualLinspeed();
update_TC();
update_axis_distance();


//-------------------------------------------------------------------------------------------------------------- MOTOR CONTROL --------------------------------------------------------------------------------------------------------------
CASE state OF
	00: //INIT STATE
	
	tstart:=TIME();
	state:=10;
	// ========================================10========================================
	10: //STANDBY STATE. 
	//wait for user inputs to transition to tension state. All motors are idle. Can edit params
	
	stop_all();
	allowInputEdits:=TRUE;
	// ========================================10========================================
	
	// ========================================11========================================
	11:
	allowInputEdits:=TRUE;
	freespin_all();
	// ========================================11========================================
	// ========================================20========================================
	20: //STANDBY WITH STANDSTILL TENSION INITAL
	//inital error check for standstill tension state
	allowInputEdits:=FALSE;
	count_enabled_motors();
	//check inputs for standstill tension
	IF standstill_tension_check() THEN
		//if error then revert to standby
		state:=10;
		hmiConnection^.tensionUI:=FALSE;
	ELSE
		state:=21;
		
	END_IF
	// ========================================20========================================
	
	// ========================================21========================================
	21://STANDBY WITH STANDSTILL TENSION
	//no movement in cable, but tension is being created. waiting on user inputs to start winding. Can edit params
	
	
	standstill_tension();
	// ========================================21========================================

	// ========================================30========================================
	30: //WINDING TENSION INITAL
	//inital error check for winding tension state.
	allowInputEdits:=FALSE;
	count_enabled_motors();
	// INPUT VALIDATION
	IF winding_check() THEN
		//if error then revert to standby
		state:=20;
		hmiConnection^.startUI:=FALSE;
		
		
		
	ELSE
		eventLogger^.fbMessage[1].Send(0);
		state:=31;
		tStart:=TIME();
	END_IF
	// ========================================30========================================
	
	// ========================================31========================================
	31: //WINDING TENSION, ACCELERATION
	//coil is currently ramping speed. can not edit params.
	
	

	
	accelerating_tension();
	determine_motor_state();
	tElapsed:=TIME() -tStart;
	
	IF winding_exit_check() THEN
	
		state:=39;
		
	ELSE
		state:=31;
	END_IF
	
	
	// ========================================31========================================
	
	// ========================================32========================================
	32: //WINDING TENSION, STEADY STATE
	//coil is in steady state. moving at constant velo with set tension. Can not edit params
	
	
	
	winding_tension();
	determine_motor_state();
	tElapsed:=TIME() -tStart;

	//check for exit conditions 
	IF winding_exit_check() THEN
		
		state:=39;
		
	ELSE
		state:=32;
	END_IF
	
	
	
	// ========================================32========================================
	
	// ========================================33========================================
	33: //WINDING TENSION, DEACCELERATION
	//coil currently decreasing speed, while maintaining. Can not edit params
	

	
	decelerating_tension();
	determine_motor_state();
	tElapsed:=TIME() -tStart;

	//check for exit conditions 
	IF winding_exit_check() THEN
		
		state:=39;
		
	ELSE
		state:=33;
	END_IF
	// ========================================33========================================
	
	// ========================================39========================================
	39: // transition state from winding => finished
		eventLogger^.fbMessage[2].Send(0);
		hmiConnection^.startUI:=FALSE;
		
		tEnd:=TIME();
		tElapsed:=tEnd -Tstart;
		
		fileReadWrite^.update_database(user:= 'TO DO figure out how to get user information',
										timeStarted:=tStart,
										timeCompleted:=tEnd,
										timeElasped:=tElapsed,
										numOfCoil:=numOfEnabledPayoff,
										lengthOCoil:=find_tape_length_used(),
										userNote:=hmiConnection^.userNote);
		fileReadWrite^.bInitWrite:=TRUE;			
		
	
		state:=40;
	// ========================================39========================================
	
	
	// ========================================40========================================
	40: //FINISHED HOLD STANDSTILL TENSION
	//cable winding finished, currently mainting tension until user input. Can not edit params
	allowInputEdits:=FALSE;
	standstill_tension();
	
	IF standstill_tension_check() THEN
		//if error then revert to standby
		state:=51;
		
	ELSE
		state:=40;
		
	END_IF
	// ========================================40========================================
	
	// ========================================41========================================
	41: //FINISHED NO TENSION
	//cable winding finished, waiting on user reset to transition to standby state. Can edit params
	//do not control tension
	stop_all();
	// ========================================41========================================
	

	// ========================================50========================================
	50:
	//exit homing state if homing is done or error.
	allowInputEdits:=FALSE;
	IF set_pos_all() THEN
		state:=10;
		hmiConnection^.homeUI:=FALSE;
	
	ELSE
		state:=50;
	END_IF
	
	
	
	
	
	// ========================================50========================================
	
	// ========================================60========================================
	60:
	//exit homing state if homing is done or error.
		allowInputEdits:=FALSE;
	IF Home() THEN
		state:=10;
		hmiConnection^.homeUI:=FALSE;
	
	ELSE
		state:=50;
	END_IF
	
	
	// ========================================60========================================
	
	
	400: //ERROR STATE
	//error on a axis preventing motor movement, or winding start. //do nothing 'till resolved
		allowInputEdits:=FALSE;
	500: //ESTOP STATE
	//triggered on estop press. can be cleared with reset
	
		hmiConnection^.tensionUI:=FALSE;
		hmiConnection^.freespinUI:=FALSE;
		hmiConnection^.startUI:=FALSE;
		allowInputEdits:=FALSE;
		estop_routine();
		
	
END_CASE
//-------------------------------------------------------------------------------------------------------------- MOTOR CONTROL --------------------------------------------------------------------------------------------------------------

//get status updates
//only calculate once very N turns in order to save resources. there also shouldnt be need to run eveyr plc cycle
	
IF (cnt MOD 10 =0) and  NOT(desiredLinspeed = 0) THEN
	etaFormattedString:=find_eta();
	progressPercent :=get_current_progress();
END_IF


//Call cyclic methods of all axies 
pickup_axis_list[1].CYLIC();

FOR i:= 1 TO GVL.MAX_PAYOFF_COUNT DO
	payoff_axis_list[i].CYLIC();
END_FOR
END_METHOD

METHOD decelerating_tension : BOOL
VAR_INPUT
END_VAR
winding_tension();
END_METHOD

METHOD determine_motor_state : BOOL
VAR_INPUT
END_VAR





VAR
	actualLinspeed : LREAL;
END_VAR
//to do . comeback on this and do a once over. not sure if this is what we want.
			
actualLinspeed:=pickup_axis_list[1].getDistToAxis()*pickup_axis_list[1].actualVelocity/57.29578;
		
//if we are below our desired
IF actualLinspeed <= 0.9*desiredLinspeed THEN
	
	state:=31;

//last turn dedicated to decelerating 
ELSIF pickup_axis_list[1].AXIS.NcToPlc.ModuloActTurns = desiredTurnCountPickup-1 THEN

	state:=33;

//if not accelerating or decelerating then we are in steady state
ELSE

	state:=32;
	
END_IF
END_METHOD

METHOD estop_routine : BOOL
VAR_INPUT
END_VAR

VAR
	i: INT;
END_VAR
//during estop, cut power to motors.

//turn power off on all axies. 
pickup_axis_list[1].MCPOWER(Axis:=pickup_axis_list[1].AXIS,ENABLE:=FALSE);

FOR i:=1 TO GVL.MAX_PAYOFF_COUNT DO
		payoff_axis_list[i].MCPOWER(Axis:=payoff_axis_list[i].AXIS,ENABLE:=FALSE);
END_FOR
END_METHOD

METHOD find_actualLinspeed : BOOL
VAR_INPUT
END_VAR
actualLinspeed:=pickup_axis_list[1].actualVelocity*pickup_axis_list[1].outerRadiusCurrent;
END_METHOD

//updates eta var
METHOD find_eta : STRING(255)
VAR
	length : LREAL; //length of straight sections in race track coil
	minutes: DINT;
	
	seconds: DINT;
	minutesString: STRING;
	secondsString: STRING;
	formattedString: STRING(255);
	tape_thicnes: LREAL :=0; //total tape thickness in meters
	i: INT;
	total_circum: LREAL;
	currentTurnCount: LREAL;
	currentCircum: LREAL;
END_VAR
VAR CONSTANT
	pi : LREAL := 4 * ATAN(1);
END_VAR
//if we are finished out put 0 seconds and exit
IF state <=59 AND state >= 50 THEN
eta:=0;
RETURN ;
END_IF

CASE pickup_axis_list[1].coilShapeID OF
	//finds eta given turn count
	//formulas are a function of circumfrence given turn count. we take the intergral of this, with respect to turn count, with the upper bound being our target turn count 
	0:
	
	tape_thicnes:=0;
	FOR i:=1 TO GVL.MAX_PAYOFF_COUNT DO
		IF payoff_axis_list[i].enabled THEN
		tape_thicnes:=tape_thicnes+payoff_axis_list[i].tape_info^[payoff_axis_list[i].tapeType].tape_depth/1000;
		END_IF
	END_FOR
	

	
	
	
	
	//finds current turn count. 
	currentTurnCount:=(pickup_axis_list[1].AXIS.NcToPlc.ModuloActPos/360+pickup_axis_list[1].AXIS.NcToPlc.ModuloActTurns);
	

	IF NOT(pickup_axis_list[1].AXIS.NcToPlc.ActVelo =0) THEN
		eta:=(desiredTurnCountPickup*360-currentTurnCount*360)/(pickup_axis_list[1].AXIS.NcToPlc.ActVelo);
	ELSE
		eta:=0;
	END_IF
	

	
	
	
	1:	
	// to do. update this monster of a formula for the race track coil. derived through calculus, which is probably correct, just now cant figure it out because i decided to write a one liner instead of splitting up
	(*
	eta:=((2*pi*racetrack_params.radius*target_turn_count_pickup+pi*tape_info.tape_depth*target_turn_count_pickup*target_turn_count_pickup+2*racetrack_params.length*target_turn_count_pickup)
		 -(2*pi*racetrack_params.radius*pickup_motor_list[1].turn_count+pi*tape_info.tape_depth*target_turn_count_pickup*pickup_motor_list[1].turn_count+2*racetrack_params.length*pickup_motor_list[1].turn_count));
		 *)
END_CASE


IF eta < 0 OR eta > 1E6 THEN
	eta:=0;
END_IF

// Convert the LREAL value to minutes and seconds
minutes := TRUNC(eta / 60);
seconds := TRUNC(eta - (minutes * 60));


// Convert the minutes and seconds to strings
minutesString := DINT_TO_STRING(minutes);

IF seconds < 10 THEN
	secondsString :=CONCAT('0', DINT_TO_STRING(seconds)) ;
ELSE
	secondsString := DINT_TO_STRING(seconds);
END_IF


// Format the final output string
find_eta := CONCAT(CONCAT('ETA: ', minutesString), CONCAT(':', secondsString));
END_METHOD

METHOD find_tape_length_used : LREAL
VAR_INPUT
END_VAR

VAR
	tape_thicnes: LREAL;
	i: INT;
	total_circum: LREAL;
END_VAR
//TO DO not sure how acurate this. i sort of stole this code from another function.

CASE pickup_axis_list[1].coilShapeID OF
	//finds eta given turn count
	//formulas are a function of circumfrence given turn count. we take the intergral of this, with respect to turn count, with the upper bound being our target turn count 
	0:
	
	tape_thicnes:=0;
	FOR i:=1 TO GVL.MAX_PAYOFF_COUNT DO
		IF payoff_axis_list[i].enabled THEN
		tape_thicnes:=tape_thicnes+payoff_axis_list[i].tape_info^[payoff_axis_list[i].tapeType].tape_depth/1000;
		END_IF
	END_FOR
	

	
	
	
	total_circum:=2*pi*desiredTurnCountPickup*pickup_axis_list[1].pancake.radius/1000 + tape_thicnes*EXPT(desiredTurnCountPickup,2)*pi;
	
	
	

	
	
	
	1:	
	// to do. update this monster of a formula for the race track coil. derived through calculus, which is probably correct, just now cant figure it out because i decided to write a one liner instead of splitting up
	(*
	eta:=((2*pi*racetrack_params.radius*target_turn_count_pickup+pi*tape_info.tape_depth*target_turn_count_pickup*target_turn_count_pickup+2*racetrack_params.length*target_turn_count_pickup)
		 -(2*pi*racetrack_params.radius*pickup_motor_list[1].turn_count+pi*tape_info.tape_depth*target_turn_count_pickup*pickup_motor_list[1].turn_count+2*racetrack_params.length*pickup_motor_list[1].turn_count));
		 *)
END_CASE



find_tape_length_used:=total_circum;
END_METHOD

METHOD freespin_all : BOOL
VAR_INPUT
END_VAR

VAR
	i: INT;
END_VAR

	pickup_axis_list[1].setFree();
		
	FOR i:=1 TO GVL.MAX_PAYOFF_COUNT DO
		
			payoff_axis_list[i].setFree();
			
		
	END_FOR
END_METHOD

METHOD general_error_check : BOOL
VAR
	i: INT;
	pickup_motor_count: INT;
	adsError : BOOL;
END_VAR
VAR_OUTPUT
	errorStatus : BOOL ;
END_VAR
VAR_IN_OUT
	errorOutput: BOOL ;
END_VAR
//Checks to see if there are any errors in a enabled axis.


pickup_axis_list[1].error_check_all();

errorStatus:=pickup_axis_list[1].AXIS.Status.Error OR pickup_axis_list[1].adsError ;
		
IF errorOutput AND pickup_axis_list[1].AXIS.Status.Error THEN
			
			ADSLOGSTR(
        		msgCtrlMask := ADSLOG_MSGTYPE_ERROR OR ADSLOG_MSGTYPE_MSGBOX,
        		msgFmtStr := 'Error occurred. Error on Pickup Axis with ID: %S',
        		strArg := UDINT_TO_STRING(pickup_axis_list[1].AXIS.Status.ErrorID)
   			 );
		
			errorOutput:=FALSE;
		
END_IF
		
IF errorOutput AND pickup_axis_list[1].adsError THEN
			
			ADSLOGSTR(
        		msgCtrlMask := ADSLOG_MSGTYPE_ERROR OR ADSLOG_MSGTYPE_MSGBOX,
        		msgFmtStr := 'Error occurred. Error in Pickup Axis FB with ID: %S ',
        		strArg := UDINT_TO_STRING(pickup_axis_list[1].adsErrorID)
   			 );
		
			errorOutput:=FALSE;
		
END_IF



FOR i:= 1 TO GVL.MAX_PAYOFF_COUNT DO
	
	payoff_axis_list[i].error_check_all();

	
		errorStatus:=errorStatus OR ((payoff_axis_list[i].AXIS.Status.Error OR payoff_axis_list[i].adsError) AND payoff_axis_list[i].enabled);
		
		IF errorOutput AND payoff_axis_list[i].AXIS.Status.Error THEN
			
			ADSLOGSTR(
        		msgCtrlMask := ADSLOG_MSGTYPE_ERROR OR ADSLOG_MSGTYPE_MSGBOX,
        		msgFmtStr := 'Error occurred. Error on Pickup Axis with ID: %S',
        		strArg := UDINT_TO_STRING(payoff_axis_list[i].AXIS.Status.ErrorID)
   			 );
		
			errorOutput:=FALSE;
		
END_IF
		
IF errorOutput AND payoff_axis_list[i].adsError THEN
			
			ADSLOGSTR(
        		msgCtrlMask := ADSLOG_MSGTYPE_ERROR OR ADSLOG_MSGTYPE_MSGBOX,
        		msgFmtStr := 'Error occurred. Error in Pickup Axis FB with ID: %S ',
        		strArg := UDINT_TO_STRING(payoff_axis_list[i].adsErrorID)
   			 );
		
			errorOutput:=FALSE;
		
END_IF
		
END_FOR
END_METHOD

METHOD general_input_check : BOOL
VAR_INPUT
	write: BOOL;
END_VAR
IF hmiConnection^.general_input_datagrid_params_list[1].tension < input_bounds.tension_low OR hmiConnection^.general_input_datagrid_params_list[1].tension > input_bounds.tension_high THEN
	general_input_check := TRUE;
	
	ADSLOGSTR(
        	msgCtrlMask := ADSLOG_MSGTYPE_ERROR OR ADSLOG_MSGTYPE_MSGBOX,
        	msgFmtStr := 'Error occurred. Tension outside of range. ',
        	strArg := ''
   		 );
	
ELSE
	
	IF write THEN
		desiredTension:=hmiConnection^.general_input_datagrid_params_list[1].tension;
	
	END_IF
END_IF

IF hmiConnection^.general_input_datagrid_params_list[1].linspeed < input_bounds.linear_speed_low OR hmiConnection^.general_input_datagrid_params_list[1].linspeed > input_bounds.linear_speed_high THEN
	general_input_check := TRUE;
	
	ADSLOGSTR(
        	msgCtrlMask := ADSLOG_MSGTYPE_ERROR OR ADSLOG_MSGTYPE_MSGBOX,
        	msgFmtStr := 'Error occurred. Linear speedc out of range.',
        	strArg := ''
   		 );
	
ELSE
	IF write THEN
		desiredLinspeed:=hmiConnection^.general_input_datagrid_params_list[1].linspeed;
	
	END_IF
	
END_IF

IF write THEN
	unwinding:=hmiConnection^.general_input_datagrid_params_list[1].unwinding;
	
END_IF
END_METHOD

METHOD get_current_progress : LREAL

VAR
	prog : LREAL;
END_VAR
IF unwinding THEN
	prog := 100-(pickup_axis_list[1].AXIS.NcToPlc.ModuloActTurns/desiredTurnCountPickup)*100;
	
ELSE
	prog := ((pickup_axis_list[1].AXIS.NcToPlc.ModuloActPos/360+pickup_axis_list[1].AXIS.NcToPlc.ModuloActTurns)/desiredTurnCountPickup)*100;

END_IF
	


IF (0 < prog AND prog < 100) THEN
	
	get_current_progress:=prog;
	
ELSIF prog > 100 THEN
	
	prog:=100;

ELSIF prog < 0 THEN
	
	prog:=0;
	
END_IF
END_METHOD

METHOD get_dist_to_axis_pickup : LREAL
VAR
	dist : LREAL;
	i: INT;
	temp: LREAL;
END_VAR
//Finds distance to axis from internal dimension and turn count vars. 

//NOTE: this only works for payoff axies. 

//output units in mm. IMPORTANT

CASE pickup_axis_list[1].coilShapeID OF
	0:
	
	CASE pickup_axis_list[1].directionB OF
		
	0: //Finds direction if motor is being unwound
	
	dist:=(pickup_axis_list[1].pancake.radius)/1000; 
	
	FOR i:=1 TO numOfEnabledPayoff DO
		IF payoff_axis_list[i].enabled THEN
			temp:=temp +(pickup_axis_list[1].axis.NcToPlc.ModuloActTurns*payoff_axis_list[i].tape_info^[payoff_axis_list[i].tapeType].tape_depth)/(1000);
		END_IF
		dist:=dist+temp;
		
	END_FOR
	1: //Finds direction if motor is being wound
	
	//to do implement directions
	
	dist:=(pickup_axis_list[1].pancake.radius)/1000; 
	
		FOR i:=1 TO numOfEnabledPayoff DO
		IF payoff_axis_list[i].enabled THEN
			temp:=temp +(pickup_axis_list[1].axis.NcToPlc.ModuloActTurns*payoff_axis_list[i].tape_info^[payoff_axis_list[i].tapeType].tape_depth)/(1000);
		END_IF
		dist:=dist+temp;
		
	END_FOR
	
	END_CASE
	
	
	
	
	
	1://TO DO. IMPLEMENT OTHER COIL IDS BESDIES PANCAKE
END_CASE
get_dist_to_axis_pickup:=dist;
END_METHOD

METHOD hmi_update : BOOL
VAR_INPUT
END_VAR

VAR
	i: INT;
END_VAR
//collection of functions to update hmi vars. 

hmiConnection^.state:=state;

update_error_status();
update_torque();
update_velocity();



hmiConnection^.overview_outputs_datagrid_list[1].pickupTurnCount:=(pickup_axis_list[1].AXIS.NcToPlc.ModuloActPos/360+pickup_axis_list[1].AXIS.NcToPlc.ModuloActTurns);
hmiConnection^.overview_outputs_datagrid_list[1].linspeed:=pickup_axis_list[1].actualVelocity*pickup_axis_list[1].outerRadiusCurrent/57.29578;




hmiConnection^.overview_outputs_datagrid_list[1].torque:=pickup_axis_list[1].actualTorque/pickup_axis_list[1].outerRadiusCurrent;

hmiConnection^.turncount_output_datagrid_list[1].pickupTC1:=(pickup_axis_list[1].AXIS.NcToPlc.ModuloActPos/360+pickup_axis_list[1].AXIS.NcToPlc.ModuloActTurns);
hmiConnection^.turncount_output_datagrid_list[1].payoffTC1:=(payoff_axis_list[1].AXIS.NcToPlc.ModuloActPos/360+payoff_axis_list[1].AXIS.NcToPlc.ModuloActTurns);
hmiConnection^.turncount_output_datagrid_list[1].payoffTC2:=(payoff_axis_list[2].AXIS.NcToPlc.ModuloActPos/360+payoff_axis_list[2].AXIS.NcToPlc.ModuloActTurns);
hmiConnection^.turncount_output_datagrid_list[1].payoffTC3:=(payoff_axis_list[3].AXIS.NcToPlc.ModuloActPos/360+payoff_axis_list[3].AXIS.NcToPlc.ModuloActTurns);


FOR i:=1 TO gvl.MAX_PAYOFF_COUNT+gvl.MAX_PICKUP_COUNT DO
	hmiConnection^.motor_info_datagrid_list[i].errorType:=axis_list[i]^.errorType;
	hmiConnection^.motor_info_datagrid_list[i].errorID:=axis_list[i]^.errorID;
	hmiConnection^.motor_info_datagrid_list[i].currentRadius:=axis_list[i]^.outerRadiusCurrent;
END_FOR
END_METHOD

METHOD home : BOOL
VAR_INPUT
END_VAR

VAR
	i: INT;
	busytemp: BOOL;
	errortemp: BOOL;
	busy: INT;
	error: INT;
END_VAR
//inital jog (so function not closed right away)
END_METHOD

METHOD INIT : BOOL
VAR_INPUT
END_VAR

VAR
	i: INT;
END_VAR
init_coil_model();
//Call cyclic methods of all axies 

pickup_axis_list[1].INIT();

pickup_axis_list[1].torqaueConstrant:=GVL.PICKUP_TORQUE_CONSTANT;
pickup_axis_list[1].ratedCurrent:=GVL.PICKUP_RATED_CURRENT;
pickup_axis_list[1].enabled:=TRUE;

pickup_axis_list[1].gearRatioNum:=10;
pickup_axis_list[1].gearRatioDen:=1;
pickup_axis_list[1].tape_info:=ADR(tape_info);

FOR i:= 1 TO GVL.MAX_PAYOFF_COUNT DO
	payoff_axis_list[i].INIT();
	payoff_axis_list[i].torqaueConstrant:=GVL.PAYOFF_TORQUE_CONSTANT;
	payoff_axis_list[i].ratedCurrent:=GVL.PAYOFF_RATED_CURRENT;
	payoff_axis_list[i].gearRatioNum:=60;
	payoff_axis_list[i].gearRatioDen:=1;
	payoff_axis_list[i].tape_info:=ADR(tape_info);
	
END_FOR

etaFormattedString := CONCAT(CONCAT('ETA: ', '0'), CONCAT(':', '0'));


axis_list[1]:=ADR(pickup_axis_list[1]);
axis_list[2]:=ADR(payoff_axis_list[1]);
axis_list[3]:=ADR(payoff_axis_list[2]);
axis_list[4]:=ADR(payoff_axis_list[3]);
END_METHOD

METHOD init_coil_model : BOOL
VAR 
	med_val : LREAL; // intermediate value 
	i :INT ;
	
	coil_type: INT:=0;
	cnt: INT :=0; //temp
END_VAR
VAR CONSTANT
	
END_VAR
//TO DO this funciton was orginall made to create a model of a non circular pickup coil shape. i would like to redo it. 

(*



	//1:
	//creates 1205 points to model a race track coil. we do this 
	cnt:=0;
	FOR i := -150 TO 150 DO
    	coil_model_base_Xcords[1][i+151]:=racetrack_params_1.radius+pickup_motor_list[1].turn_count*tape_info.tape_depth;
		coil_model_base_Ycords[1][i+151]:=i;
		
		
	END_FOR;
	FOR i := -150 TO 150 DO
    	coil_model_base_Xcords[1][i+452]:=-(coil_shape_params.radius+pickup_motor_list[1].turn_count*tape_info.tape_depth);
		coil_model_base_Ycords[1][i+452]:=i;
	
	END_FOR;
	FOR i := -150 TO 150 DO
		med_val:=(pi/300)*i+pi;
		
		
    	coil_model_base_Xcords[1][i+753]:=(coil_shape_params.radius+pickup_motor_list[1].turn_count*tape_info.tape_depth)*SIN(med_val);
		coil_model_base_Ycords[1][i+753]:=-1*coil_shape_params.length*COS(med_val);
	
	END_FOR;
	FOR i := -150 TO 150 DO
		med_val:=(pi/300)*i;
		
		
    	coil_model_base_Xcords[1][i+904]:=(coil_shape_params.radius+pickup_motor_list[1].turn_count*tape_info.tape_depth)*SIN(med_val);
		coil_model_base_Ycords[1][i+904]:=coil_shape_params.length*COS(med_val);
	
	END_FOR;
	 
*)
END_METHOD

METHOD input_update : BOOL
VAR_INPUT
	general : BOOL ;
	pickup : BOOL ;
	payoff : BOOL ;
END_VAR



VAR
	
	//chooses which inputs we will update.         
	i: INT;
END_VAR
//NOT NEEDED ANYMORE
(*


//Updates internal winding control variables with HMI inputs. 
IF pickup THEN
	pickup_axis_list[1].coilShapeID:=hmiConnection^.pickup_input_datagrid_params_list[1].coil_shape;
	desiredTurnCountPickup:=hmiConnection^.pickup_input_datagrid_params_list[1].turn_count;
END_IF

IF payoff THEN
	FOR i:= 1 TO GVL.MAX_PAYOFF_COUNT DO
		payoff_axis_list[i].enabled:=hmiConnection^.payoff_input_datagrid_params_list[i].enabled;
	IF payoff_axis_list[i].enabled THEN
		payoff_axis_list[i].pancake.radius:=hmiConnection^.payoff_input_datagrid_params_list[i].outer_dia;
		
	
	END_IF
	
	END_FOR
END_IF

IF general THEN
	desiredLinspeed:=hmiConnection^.general_input_datagrid_params_list[1].linspeed;
	desiredTension:=hmiConnection^.general_input_datagrid_params_list[1].tension;
	unwinding:=hmiConnection^.general_input_datagrid_params_list[1].unwinding;
	
	pickup_axis_list[1].directionB:=BOOL_TO_INT(unwinding);
	
	FOR i:= 1 TO GVL.MAX_PAYOFF_COUNT DO
		payoff_axis_list[i].directionB:=BOOL_TO_INT(unwinding);

	END_FOR
END_IF

*)
END_METHOD

METHOD payoff_input_check : BOOL
VAR_INPUT
END_VAR

VAR_input
	write: BOOL;
END_VAR
VAR
	i: INT;
END_VAR
 FOR i:= 1 TO GVL.MAX_PAYOFF_COUNT DO
	
	IF write THEN
		payoff_axis_list[i].enabled:=hmiConnection^.payoff_input_datagrid_params_list[i].enabled;
		payoff_axis_list[i].tapeType:=hmiConnection^.payoff_input_datagrid_params_list[i].tape_type;
		payoff_axis_list[i].pancake.radius:=hmiConnection^.payoff_input_datagrid_params_list[i].radius;
	END_IF

	
END_FOR
END_METHOD

METHOD pickup_input_check : BOOL
VAR_INPUT
	write : BOOL ;
END_VAR
IF hmiConnection^.pickup_input_datagrid_params_list[1].turn_count < input_bounds.turn_count_pickup_low OR hmiConnection^.pickup_input_datagrid_params_list[1].turn_count > input_bounds.turn_count_pickup_high THEN
	pickup_input_check := TRUE;
	
	ADSLOGSTR(
        	msgCtrlMask := ADSLOG_MSGTYPE_ERROR OR ADSLOG_MSGTYPE_MSGBOX,
        	msgFmtStr := 'Error occurred. Pickup turncount outside of range.',
        	strArg := ''
   		 );
	
ELSE
	
	IF write THEN
		desiredTurnCountPickup:=hmiConnection^.pickup_input_datagrid_params_list[1].turn_count;
	END_IF

	
	
	
END_IF
END_METHOD

METHOD read_status : BOOL
VAR_INPUT
END_VAR

VAR
	i: INT;
END_VAR
 //updates status of all axises, pickup and payoff

pickup_axis_list[1].Axis.ReadStatus();


FOR i:= 1 TO GVL.MAX_PAYOFF_COUNT DO
	payoff_axis_list[i].AXIS.ReadStatus();
END_FOR
END_METHOD

METHOD reset : BOOL
VAR_INPUT
END_VAR

VAR
	i: INT;
END_VAR
state := 10;
progressPercent:=0;

fileReadWrite^.reset();

// reset axis's, clear errors
pickup_axis_list[1].reset();
		
pickup_axis_list[1].SoEReset(axis:=pickup_axis_list[1].AXIS,Execute:=FALSE);

pickup_axis_list[1].SoEReset(axis:=pickup_axis_list[1].AXIS,Execute:=TRUE);

FOR i:=1 TO GVL.MAX_PAYOFF_COUNT DO
		
			payoff_axis_list[i].reset();
			
		
END_FOR
END_METHOD

METHOD set_pos_all : BOOL
VAR_INPUT
END_VAR

VAR

	i: INT;
	busy : BOOL :=FALSE;
	busytemp : BOOL := FALSE;
	error : BOOL:= FALSE;
	errorTemp : BOOL := FALSE;
END_VAR
//to do . bug where after a failed winding attemp, users need to press button one more time inorder for command to run. coming back to this later

//function to set pos of all motors to 0

//turn power off on all axies. need for set pos function
pickup_axis_list[1].MCPOWER(Axis:=pickup_axis_list[1].AXIS,ENABLE:=FALSE);

FOR i:=1 TO GVL.MAX_PAYOFF_COUNT DO
	IF payoff_axis_list[i].enabled THEN
			
		payoff_axis_list[i].MCPOWER(Axis:=payoff_axis_list[i].AXIS,ENABLE:=FALSE);
	END_IF
END_FOR 




//set pos, repeat till not busy. 
REPEAT
	
	//set pos of pickup
	pickup_axis_list[1].MCPOS(Axis:=pickup_axis_list[1].Axis,Execute:=TRUE,Position:=0,MODE:=FALSE,busy=>busytemp,Error=>errortemp);
	busy:= busy AND busytemp;
	error:= error AND errorTemp;


//set pos of payoff
	FOR i:=1 TO GVL.MAX_PAYOFF_COUNT DO
		IF payoff_axis_list[i].enabled THEN
			
			payoff_axis_list[i].MCPOS(Axis:=payoff_axis_list[i].Axis,Execute:=TRUE,Position:=0,MODE:=FALSE,busy=>busytemp,Error=>errortemp);
			busy:=busy AND busytemp;
			error:= error AND errorTemp;
		END_IF
	END_FOR 


//exit condition	
UNTIL 
//exit when all axies are no longer busy
NOT BUSY
END_REPEAT

pickup_axis_list[1].MCPOS(Axis:=pickup_axis_list[1].Axis, Execute:=TRUE,Position:=0,mode:=FALSE);




//turn power off on all axies. 
pickup_axis_list[1].MCPOWER(Axis:=pickup_axis_list[1].AXIS,ENABLE:=TRUE);
pickup_axis_list[1].MCPOS(Axis:=pickup_axis_list[1].Axis,Execute:=FALSE,Position:=0,MODE:=FALSE,busy=>busytemp,Error=>errortemp);

FOR i:=1 TO GVL.MAX_PAYOFF_COUNT DO
	IF payoff_axis_list[i].enabled THEN
		payoff_axis_list[i].MCPOWER(Axis:=payoff_axis_list[i].AXIS,ENABLE:=TRUE);
		payoff_axis_list[i].MCPOS(Axis:=payoff_axis_list[i].Axis,Execute:=FALSE,Position:=0,MODE:=FALSE,busy=>busytemp,Error=>errortemp);
			busy:=busy AND busytemp;
	END_IF		
END_FOR 
set_pos_all:=NOT ERROR;
END_METHOD

METHOD standstill_tension : BOOL
VAR_INPUT
	
END_VAR

VAR
	
	i: INT;
END_VAR
//creates tension in tape, but does not move the tape.

//set torque to force times number of payoff motors enabled. 

pickup_axis_list[1].torque:=((desiredTension*numOfEnabledPayoff* pickup_axis_list[1].outerRadiusCurrent)/2)+GVL.MIN_THRESHOLD_TORQUE;
	
//TO DO need to find what to set these to. might be too low. 
pickup_axis_list[1].velocityLimitLow:=50;
pickup_axis_list[1].velocityLimitHigh:=50;
	
	
pickup_axis_list[1].setTorque();
	
	
FOR i:=1 TO GVL.MAX_PAYOFF_COUNT DO
	IF payoff_axis_list[i].enabled THEN
		payoff_axis_list[i].setTorque();
		
		payoff_axis_list[i].velocityLimitLow:=-70;
		payoff_axis_list[i].velocityLimitHigh:=-70;
		payoff_axis_list[i].torque:=-1*((desiredTension*	payoff_axis_list[i].outerRadiusCurrent/2)+GVL.MIN_THRESHOLD_TORQUE)-5;
			
	END_IF
END_FOR
END_METHOD

METHOD standstill_tension_check : BOOL
VAR_OUTPUT

END_VAR
VAR
	input_bounds : input_bounds; //struct defining input bounds
	i: INT; //counter
	
	
	payoffEnableCheck :BOOL :=FALSE; //var to hold payoff enable var
END_VAR
//check to see if HMI vars are valid for stand still tension before winding. outputs true if there was an error.

//PICKUP AXIS CHECKS
payoff_input_check(write:=TRUE);

IF hmiConnection^.general_input_datagrid_params_list[1].tension < input_bounds.tension_low OR hmiConnection^.general_input_datagrid_params_list[1].tension > input_bounds.tension_high THEN
	standstill_tension_check := TRUE;
	
	ADSLOGSTR(
        	msgCtrlMask := ADSLOG_MSGTYPE_ERROR OR ADSLOG_MSGTYPE_MSGBOX,
        	msgFmtStr := 'Error occurred. Tension outside of range. Unable to start tension',
        	strArg := ''
   		 );
	
ELSE
	desiredTension:=hmiConnection^.general_input_datagrid_params_list[1].tension;
	
END_IF

//PAYOFF AXIS CHECKS

FOR i:= 1 TO GVL.MAX_PAYOFF_COUNT DO
	payoffEnableCheck:=payoffEnableCheck OR hmiConnection^.payoff_input_datagrid_params_list[i].enabled;
	

	
END_FOR


IF NOT payoffEnableCheck THEN
	standstill_tension_check := TRUE;
	
	ADSLOGSTR(
        	msgCtrlMask := ADSLOG_MSGTYPE_ERROR OR ADSLOG_MSGTYPE_MSGBOX,
        	msgFmtStr := 'Error occurred. At least one payoff motor needs to be enabled',
        	strArg := ''
   		 );

END_IF
END_METHOD

METHOD stop_all : BOOL
VAR_INPUT
END_VAR

VAR
	i: INT;
END_VAR

	pickup_axis_list[1].setStop();
		
	FOR i:=1 TO GVL.MAX_PAYOFF_COUNT DO
		
			payoff_axis_list[i].setStop();
			
		
	END_FOR
END_METHOD

METHOD transfer_hmi_vars : BOOL
VAR_INPUT
END_VAR

VAR
	i: INT;
END_VAR
//transfer vars from hmi to windingcontrol

//general
desiredTension:=hmiConnection^.general_input_datagrid_params_list[1].tension;

desiredLinspeed:=hmiConnection^.general_input_datagrid_params_list[1].linspeed;

unwinding:=hmiConnection^.general_input_datagrid_params_list[1].unwinding;

//pickup

desiredTurnCountPickup:=hmiConnection^.pickup_input_datagrid_params_list[1].turn_count;
pickup_axis_list[1].coilShapeID:=hmiConnection^.pickup_input_datagrid_params_list[1].coil_shape;
pickup_axis_list[1].pancake.radius:=hmiConnection^.pickup_pancake_input_datagrid_params_list[1].radius;
//payoff
 FOR i:= 1 TO GVL.MAX_PAYOFF_COUNT DO
	

	payoff_axis_list[i].enabled:=hmiConnection^.payoff_input_datagrid_params_list[i].enabled;
	payoff_axis_list[i].tapeType:=hmiConnection^.payoff_input_datagrid_params_list[i].tape_type;
	
	payoff_axis_list[i].pancake.radius:=hmiConnection^.payoff_input_datagrid_params_list[i].radius;
		
END_FOR
END_METHOD

METHOD turncount_check : BOOL
VAR_INPUT
END_VAR

VAR
	i: INT;
	temp: LREAL;
	ext: BOOL;
END_VAR
//checks to see if inputed turncount will result in a outer radius over max
ext:=FALSE;


dist:=(pickup_axis_list[1].pancake.radius)/1000; 
	
	FOR i:=1 TO numOfEnabledPayoff DO
		IF payoff_axis_list[i].enabled THEN
			temp:=temp + ( desiredTurnCountPickup  *payoff_axis_list[i].tape_info^[payoff_axis_list[i].tapeType].tape_depth)/(1000);
		END_IF
		dist:=dist+temp;
		
	END_FOR


//max outer radius check
IF dist*1000 >= GVL.MAX_PICKUP_RADIUS THEN
			
	ADSLOGDINT(msgCtrlMask := ADSLOG_MSGTYPE_HINT OR ADSLOG_MSGTYPE_MSGBOX, msgFmtStr := 'Winding stopped, calculated final radius above maximum radius limit, please lower turncount. Pickup Axis: %d', dintArg := 1);
	
	ext :=TRUE;
		
END_IF


turncount_check:=ext;
END_METHOD

METHOD update_axis_distance : BOOL
VAR_INPUT
END_VAR

VAR
	i: INT;
END_VAR
pickup_axis_list[1].outerRadiusCurrent:=get_dist_to_axis_pickup();

FOR i:=1 TO gvl.MAX_PAYOFF_COUNT DO
	IF payoff_axis_list[i].enabled THEN
		payoff_axis_list[i].outerRadiusCurrent:=payoff_axis_list[i].getDistToAxis();
	END_IF
END_FOR
END_METHOD

METHOD update_error_status : BOOL
VAR_INPUT
END_VAR

VAR
	i: INT;
	
END_VAR
hmiConnection^.output_error_datagrid_list[0].errorStatus:=pickup_axis_list[1].AXIS.Status.Error;
hmiConnection^.output_error_datagrid_list[0].errorID:=pickup_axis_list[1].AXIS.Status.ErrorID;

hmiConnection^.motor_state_datagrid_list[0].state:=pickup_axis_list[1].state;

FOR i:= 1 TO GVL.MAX_PAYOFF_COUNT DO
	hmiConnection^.output_error_datagrid_list[i].errorStatus:=payoff_axis_list[i].AXIS.Status.Error;
	hmiConnection^.output_error_datagrid_list[i].errorID:=payoff_axis_list[i].AXIS.Status.ErrorID;
	
	hmiConnection^.motor_state_datagrid_list[i].state:=payoff_axis_list[i].state;
	
END_FOR
END_METHOD

METHOD update_TC : BOOL
VAR_INPUT
END_VAR


target_turn_count:=desiredTurnCountPickup;
END_METHOD

METHOD update_torque : BOOL
VAR_INPUT
END_VAR

VAR
	i: INT;
END_VAR
//update act ual torque values ofc motors. send these values to HMI

pickup_axis_list[1].getTorque();
hmiConnection^.torque[1]:=pickup_axis_list[1].actualTorque;
hmiConnection^.motor_info_datagrid_list[1].torque:=hmiConnection^.torque[1];

FOR i:= 1 TO GVL.MAX_PAYOFF_COUNT DO
	payoff_axis_list[i].getTorque();
	hmiConnection^.torque[i+1]:=payoff_axis_list[i].actualTorque;
	hmiConnection^.motor_info_datagrid_list[i+1].torque:=payoff_axis_list[i].actualTorque;;
END_FOR
END_METHOD

METHOD update_velocity : BOOL
VAR_INPUT
END_VAR

VAR
	i: INT;
END_VAR
//update act ual torque values ofc motors. send these values to HMI


hmiConnection^.rpm[1]:=pickup_axis_list[1].actualVelocity;
hmiConnection^.rpm[2]:=payoff_axis_list[1].actualVelocity;
hmiConnection^.rpm[3]:=payoff_axis_list[2].actualVelocity;
hmiConnection^.rpm[4]:=payoff_axis_list[3].actualVelocity;


hmiConnection^.motor_info_datagrid_list[1].speed:=hmiConnection^.rpm[1];
hmiConnection^.motor_info_datagrid_list[2].speed:=hmiConnection^.rpm[2];
hmiConnection^.motor_info_datagrid_list[3].speed:=hmiConnection^.rpm[3];
hmiConnection^.motor_info_datagrid_list[4].speed:=hmiConnection^.rpm[4];
END_METHOD

METHOD winding_check : BOOL
VAR_INPUT
END_VAR
winding_check:= winding_check OR turncount_check();
END_METHOD

METHOD winding_exit_check : BOOL
VAR_INPUT
END_VAR

VAR
	ext : BOOL :=FAlse;
	i: INT;
	ste : INT :=-1;
END_VAR
//Checks to see if various conditions are met to exit

//turn count condition.

IF pickup_axis_list[1].AXIS.NcToPlc.ModuloActTurns >= target_turn_count THEN

	
	ADSLOGSTR(msgCtrlMask := ADSLOG_MSGTYPE_HINT OR ADSLOG_MSGTYPE_MSGBOX, msgFmtStr := 'Winding stopped, pickup turn count reached', strArg:= '');
	ADSLOGSTR(msgCtrlMask := ADSLOG_MSGTYPE_HINT OR ADSLOG_MSGTYPE_LOG, msgFmtStr := 'Winding stopped, pickup turn count reached', strArg:= '');
	ext := TRUE;
	
END_IF

//inner radius reached check
IF pickup_axis_list[1].outerRadiusCurrent*0.99*1000 <= GVL.MIN_MOUNT_RADIUS THEN
			
	ADSLOGDINT(msgCtrlMask := ADSLOG_MSGTYPE_HINT OR ADSLOG_MSGTYPE_MSGBOX, msgFmtStr := 'Winding stopped, calculated current radius dropped below inner radius. PICKUP AXIS ID: %d', dintArg := 1);
	ADSLOGSTR(msgCtrlMask := ADSLOG_MSGTYPE_HINT OR ADSLOG_MSGTYPE_LOG, msgFmtStr := 'Winding stopped, calculated current radius dropped below inner radius. PICKUP AXIS ID: %S', strArg := INT_TO_STRING(1));
	ext :=TRUE;
		
END_IF

FOR i:=1 TO GVL.MAX_PAYOFF_COUNT DO
	IF payoff_axis_list[i].enabled THEN
		IF payoff_axis_list[i].outerRadiusCurrent*0.99*1000 <= GVL.MIN_MOUNT_RADIUS THEN
			
			ADSLOGDINT(msgCtrlMask := ADSLOG_MSGTYPE_HINT OR ADSLOG_MSGTYPE_MSGBOX, msgFmtStr := 'Winding stopped, calculated current radius dropped below inner radius. PAYOFF AXIS ID: %d', dintArg := i);
			ADSLOGSTR(msgCtrlMask := ADSLOG_MSGTYPE_HINT OR ADSLOG_MSGTYPE_LOG, msgFmtStr := 'Winding stopped, calculated current radius dropped below inner radius. PAYOFF AXIS ID: %S', strArg := INT_TO_STRING(i));
	ext :=TRUE;
		
		END_IF
	
	END_IF
END_FOR

//max outer radius check
IF pickup_axis_list[1].outerRadiusCurrent*1.01*1000 >= GVL.MAX_PICKUP_RADIUS THEN
			
	ADSLOGDINT(msgCtrlMask := ADSLOG_MSGTYPE_HINT OR ADSLOG_MSGTYPE_MSGBOX, msgFmtStr := 'Winding stopped, calculated current radius raised above max outer radius. PICKUP AXIS ID: %d', dintArg := 1);
	ADSLOGSTR(msgCtrlMask := ADSLOG_MSGTYPE_HINT OR ADSLOG_MSGTYPE_LOG, msgFmtStr := 'Winding stopped, calculated current radius raised above max outer radius. PICKUP AXIS ID: %S', strArg := INT_TO_STRING(1));
	ext :=TRUE;
		
END_IF

FOR i:=1 TO GVL.MAX_PAYOFF_COUNT DO
	IF payoff_axis_list[i].enabled THEN
		IF payoff_axis_list[i].outerRadiusCurrent*1.01*1000 >= GVL.MAX_PAYOFF_RADIUS THEN
			
			ADSLOGDINT(msgCtrlMask := ADSLOG_MSGTYPE_HINT OR ADSLOG_MSGTYPE_MSGBOX, msgFmtStr := 'Winding stopped, calculated current radius raised above max outer radius. PAYOFF AXIS ID: %d', dintArg := i);
	
	ext :=TRUE;
		
		END_IF
	
	END_IF
END_FOR

winding_exit_check:=ext;
END_METHOD

METHOD winding_tension : BOOL
VAR_INPUT
END_VAR

VAR
	i: INT;
	
	desiredVelocity : LREAL;
	pickupLinspeed: LREAL;
	adjustedVelocity: LREAL;
	
END_VAR
VAR CONSTANT
	PERCENT_DIFFERENCE: LREAL := 1.1;
END_VAR
IF unwinding THEN
	//to do update with unwinding feature
	
	//do nothing, not implemneted yet. 
ELSE
	


	pickup_axis_list[1].torque:=desiredTension*numOfEnabledPayoff * get_dist_to_axis_pickup()+GVL.MIN_THRESHOLD_TORQUE;
	
	//TO DO . need to confirm these are correct
	//how i envison the limits to function is that the pickup side will gradually ramp up speed until we hit the upper velocity limit. we could maybe have no limits and just have only torque control
	//will need testing. 
	pickup_axis_list[1].velocityLimitLow:=0;
	pickup_axis_list[1].velocityLimitHigh:=(desiredLinspeed/pickup_axis_list[1].outerRadiusCurrent)*57.29578 ;
	
	pickup_axis_list[1].setTorque();
	
	pickupLinspeed:=pickup_axis_list[1].AXIS.NcToPlc.ActVelo*pickup_axis_list[1].outerRadiusCurrent/57.29578;
	
	
	
	FOR i:=1 TO GVL.MAX_PAYOFF_COUNT DO
		IF payoff_axis_list[i].enabled THEN
		
			
			
			
			payoff_axis_list[i].setVelocity();
			dist:=payoff_axis_list[i].outerRadiusCurrent;
		
			//find the velocity (degree/s) to acheive our desired linear speed, and the linear speed at pickup motor. 
			desiredVelocity:=(desiredLinspeed/payoff_axis_list[i].outerRadiusCurrent)*57.29578 ;
			adjustedVelocity:=(pickupLinspeed/payoff_axis_list[i].outerRadiusCurrent)*57.29578;
			
			
			
			//sets payoff axis to half way point between target linspeed and the actual linspeed.
			//how i envison this to function, is that while pickup side is at a low speed, the payoff side will also work at a lower speed,
			//which gives the pickup time to catch up in speed. right now i do this by just averaging desired speed and actual speed,
			//this could maybe he handled in a better way, so i will leave a TO DO 
			payoff_axis_list[i].velocity:=(0.05*desiredVelocity+adjustedVelocity*0.95);
			
			
			
		END_IF
	END_FOR 
END_IF
END_METHOD

END_FUNCTION_BLOCK

// ---- POUs/FB_EventLogger.TcPOU
FUNCTION_BLOCK FB_EventLogger
VAR
	fbMessage : ARRAY[0..GVL.MAX_EVENT_SIZE] OF FB_TcMessage; ///array of all possible events
END_VAR

METHOD CYCLIC : BOOL
VAR_INPUT
END_VAR
END_METHOD

METHOD INIT : BOOL
VAR_INPUT
END_VAR
//initlize event log messages
fbMessage[0].CreateEx(TC_Events.PLC_events.INIT, 0);
fbMessage[1].CreateEx(TC_Events.PLC_events.WindingStarted, 0);
fbMessage[2].CreateEx(TC_Events.PLC_events.WindingExitTC, 0);
fbMessage[3].CreateEx(TC_Events.PLC_events.InvalidInputs, 0);
fbMessage[4].CreateEx(TC_Events.PLC_events.WindingExitUser, 0);
fbMessage[5].CreateEx(TC_Events.PLC_events.AxisErrorState, 0);
fbMessage[6].CreateEx(TC_Events.PLC_events.WindingPaused, 0);
fbMessage[7].CreateEx(TC_Events.PLC_events.WindingExitUser, 0);
fbMessage[8].CreateEx(TC_Events.PLC_events.HomingError, 0);
fbMessage[9].CreateEx(TC_Events.PLC_events.ESTOP,0);




fbMessage[0].Send(0);
END_METHOD

END_FUNCTION_BLOCK

// ---- POUs/FB_fileReadWrite.TcPOU
FUNCTION_BLOCK FB_fileReadWrite

VAR_IN_OUT
	
END_VAR
VAR_OUTPUT
	bInProgress		: BOOL:=FALSE;
END_VAR
VAR_INPUT
	bInitWrite		: BOOL := FALSE;(* Rising edge starts program execution *)
	bwrite			: BOOL;
	 bStartTiming : BOOL;
    bStopTiming : BOOL;
END_VAR

VAR
	bTempb			:bool;
	
	
	sNetId			: T_AmsNetId := '';	(* TwinCAT system network address *)
	sFileRoot		: T_MaxString := 'C:\Users\nbung\Documents\TcXaeShell\CoilWindingMachine\CoilWindingHMI\LOG';
	sFilePath		: T_MaxString := '\';
	newsFilePath 	:  T_MaxString := '\';
	sFileName		: T_MaxString := '';(* CSV destination file path and name *) 
	sCSVLine		: T_MaxString := '';(* Single CSV text line (row, record), we are using string as record buffer (your are able to see created fields) *)
	sCSVField		: T_MaxString := '';(* Single CSV field value (column, record field) *)
	bBusy			: BOOL;
	bError			: BOOL;
	nErrId			: UDINT;
	nRow	 		: UDINT 	:= 0;(* Row number (record) *)
	nColumn			: UDINT 	:= 0;(* Column number (record field) *)
	hFile			: UINT		:= 0;(* File handle of the source file *)
	step			: DWORD 	:= 0;
	stepCheck		: DWORD 	:= 0;
	stepDel: INT;
	
	
	startTime : TIMESTRUCT;
    endTime : TIMESTRUCT;
    elapsedTime : TIME;
	fbTimer   : FB_LocalSystemTime := ( bEnable := TRUE, dwCycle := 1 );
	fbFileOpen		: FB_FileOpen;(* Opens file *)
	fbFileClose		: FB_FileClose;(* Closes file *)
	fbFilePuts		: FB_FilePuts;(* Writes one record (line) *)
	fbFileDelete	: FB_FileDelete;(* deletes a file*)
	fbWriter		: FB_CSVMemBufferWriter;(* Helper function block used to create CSV data bytes (single record line) *)
	bDone			: BOOL;
	bCheck          : BOOL;
	bValidPath		: BOOL;
	bDelete			: BOOL;
	
		testdatabase		: ARRAY[0..GVL.MAX_CSV_ROWS, 0..GVL.MAX_CSV_COLUMNS ] OF STRING(GVL.MAX_CSV_FIELD_LENGTH) :=[ 
	'User: ', 'TestUser',
	'Time Started: ', 'N/A', 
	'Time Completed: ', 'N/A',
	'Time Elapsed: ', 'N/A', 
	'Number OF coils: ', 'N/A',
	'Length of coil used: ', 'N/A',
	'User Note: ', 'This is a note from the user. should be last'];
	
	database		: ARRAY[0..GVL.MAX_CSV_ROWS, 0..GVL.MAX_CSV_COLUMNS ] OF STRING(GVL.MAX_CSV_FIELD_LENGTH) :=[ 
	'User: ', 'TestUser',
	'Time Started: ', 'N/A', 
	'Time Completed: ', 'N/A',
	'Time Elapsed: ', 'N/A', 
	'Number OF coils: ', 'N/A',
	'Length of coil used: ', 'N/A',
	'User Note: ', 'This is a note from the user. should be last'];
	//system time
	
END_VAR

METHOD checkFile : BOOL
VAR_INPUT
END_VAR


VAR
	tempString: STRING(255);
END_VAR
CASE stepCheck OF
	//Waiting for rising edge of writeFile Variable. standby state
	0:
		IF bCheck  THEN
			bDone	:= FALSE;
			bCheck 	:= FALSE;
			bBusy 	:= TRUE;
			bError	:= FALSE;
			nErrId	:= 0;
			hFile	:= 0;
			nRow	:= 0;
			nColumn	:= 0;
			stepCheck 	:= 1;
			
		END_IF
		
	//open file
	1:
	
		tempString := CONCAT('LOG-',WORD_TO_STRING(fbTimer.systemTime.wYear) );
		tempString := CONCAT(tempString, '-');
		tempString := CONCAT(tempString, WORD_TO_STRING(fbTimer.systemTime.wMonth));
		tempString := CONCAT(tempString, '-');
		tempString := CONCAT(tempString, WORD_TO_STRING(fbTimer.systemTime.wDay));
		tempString := CONCAT(tempString, '-');
		tempString := CONCAT(tempString, WORD_TO_STRING(fbTimer.systemTime.wHour));
		tempString := CONCAT(tempString, '-');
		tempString := CONCAT(tempString, WORD_TO_STRING(fbTimer.systemTime.wMinute));
		sFileName := tempString;
		
	//	findAndReplace(pSrcString:=ADR(sFilePath),pDeleteString:=ADR('/'),pInsertString:=ADR('\'),pDstString:=ADR(newsFilePath),nDstsize:=255);
		newsFilePath := CONCAT(sFileRoot,sFilePath);
	
		tempString := CONCAT(newsFilePath,'\'); 
		sFileName := CONCAT(tempString,sFileName);
		sFileName := CONCAT(sFileName, '.csv');
		//sFileName:='C:\Users\nbung\Downloads\new.csv';
	
	
		fbFileOpen(bExecute:=FALSE);	
		fbFileOpen(bExecute:=TRUE,
					nmode:=FOPEN_MODEWRITE,
					sPathName:=sFileName,
					ePath:=PATH_GENERIC,
					sNetId:='',
					tTimeout:=T#5S,); 
		
		stepCheck := 2;
		
		
	//wait untill we are finished opening the text file. 
	2:
		fbFileOpen( bExecute := FALSE, bError => bError, nErrID => nErrID, hFile => hFile );
		IF NOT fbFileOpen.bBusy THEN
			
			IF NOT fbFileOpen.bError THEN
				
				stepCheck := 100;
				bValidPath:=TRUE;
				bDelete :=TRUE;
				
				
		ELSE(* Error: could not create file *)
				stepCheck := 100;
				bValidPath:=FALSE;
				bError:=TRUE;
				
				  ADSLOGSTR(msgCtrlMask := ADSLOG_MSGTYPE_ERROR OR ADSLOG_MSGTYPE_MSGBOX,
                  msgFmtStr := 'Error Occured. Unable to start winding while not in tension state',
                  strArg := '');
				
				
			END_IF
		END_IF

		
	//close file
		10:
		fbFileClose( bExecute := FALSE );
		fbFileClose( sNetId := sNetId, hFile := hFile, bExecute := TRUE );
		stepCheck := 11;
	
	11:(* Wait until close not busy *)
		fbFileClose( bExecute := FALSE, bError => bError, nErrID => nErrID );
		IF ( NOT fbFileClose.bBusy ) THEN
			hFile := 0;
			stepCheck := 100;
		END_IF
	100: (* Error or ready step => cleanup *)
		IF ( hFile <> 0 ) THEN
			stepCheck := 10; (* Close the source file *)
		ELSE
			bBusy := FALSE;
			stepCheck := 0;	(* Ready *)
		END_IF
		
END_CASE
END_METHOD

METHOD CYCLIC : BOOL
VAR_INPUT
END_VAR

VAR

t : DATE_AND_TIME ;
END_VAR
fbTimer(bEnable := TRUE, dwCycle := 1 );

//if bInitWrite is selected, then
//check if path is valid, then
//delete temporary file, then
//update data base, then
//write file, then

IF bInitWrite THEN
	bCheck:=TRUE;
	bInitWrite:=FALSE;
END_IF

IF bStartTiming AND NOT bInProgress THEN
    startTime:=fbTimer.systemTime;
    bStartTiming := FALSE;
	bInProgress:= TRUE;
END_IF

// Stop timing and calculate elapsed time
IF bStopTiming THEN
   endTime:=fbTimer.systemTime;
  
    // Calculate elapsed time in milliseconds
  
    bStopTiming := FALSE;
	bInProgress :=FALSE;
END_IF

fileWrite();
checkFile();
fileDelete();
END_METHOD

METHOD fileDelete : BOOL
VAR_INPUT
END_VAR

VAR
	
END_VAR
CASE stepDel OF
	//Waiting for rising edge of writeFile Variable. standby state
	0:
		IF bDelete AND NOT bBusy THEN
			bDone	:= FALSE;
			bDelete 	:= FALSE;
			bBusy 	:= TRUE;
			bError	:= FALSE;
			nErrId	:= 0;
			hFile	:= 0;
			
			stepDel 	:= 1;
		END_IF
		
	//open file
	1:
		fbFileDelete(bExecute:=FALSE);
			fbFileDelete(bExecute:=TRUE,	
						sPathName:=sFileName,
						sNetId:='',
						tTimeout:=T#5S,);
		stepDel := 2;
	//wait untill we are finished opening the text file. 
	2:
			fbFileDelete( bExecute := FALSE, bError => bError, nErrID => nErrID );
			IF NOT fbFileDelete.bBusy THEN
			
				IF NOT fbFileDelete.bError THEN
					bDone:=TRUE;
					stepDel :=100;
					
				ELSE(* Error: could not create file *)
				stepDel := 100;
				bValidPath:=FALSE;
				bError:=TRUE;
					
				END_IF
			END_IF
	
	10:
		fbFileClose( bExecute := FALSE );
		fbFileClose( sNetId := sNetId, hFile := hFile, bExecute := TRUE );
		stepDel := 11;
	
	11:(* Wait until close not busy *)
		fbFileClose( bExecute := FALSE, bError => bError, nErrID => nErrID );
		IF ( NOT fbFileClose.bBusy ) THEN
			hFile := 0;
			stepDel := 100;
		END_IF
		
	100: (* Error or ready step => cleanup *)
		bDone:=TRUE;
		IF ( hFile <> 0 ) THEN
			stepDel := 10; (* Close the source file *)
		ELSE
			bBusy := FALSE;
			
			bwrite:= NOT berror;
			stepDel := 0;	(* Ready *)
		END_IF
END_CASE
END_METHOD

METHOD fileWrite : BOOL
VAR_INPUT
END_VAR

VAR
 tempString   : STRING;
 

 
 
 nDstsize : UDINT;
END_VAR
CASE step OF
	//Waiting for rising edge of writeFile Variable. standby state
	0:
	
		IF  bValidPath AND bWrite  THEN
			bCheck	:= FALSE;
			bDone	:= FALSE;
			bWrite 	:= FALSE;
			bBusy 	:= TRUE;
			bError	:= FALSE;
			nErrId	:= 0;
			hFile	:= 0;
			nRow	:= 0;
			nColumn	:= 0;
			step 	:= 1;
		END_IF
	
		
	//open file
	1:
		
		
		
	
		fbFileOpen(bExecute:=FALSE);
		fbFileOpen( sNetId := sNetId,
					sPathName := sFileName, 
					nMode := FOPEN_MODEWRITE OR FOPEN_MODETEXT,(* Open file in TEXT mode! *)
					ePath := PATH_GENERIC,
					bExecute := TRUE );
		step := 2;
	//wait untill we are finished opening the text file. 
	2:
		fbFileOpen( bExecute := FALSE, bError => bError, nErrID => nErrID, hFile => hFile );
		IF NOT fbFileOpen.bBusy THEN
			IF NOT fbFileOpen.bError THEN
				step := 3;
			ELSE(* Error: file not found? *)
				step := 100;
			END_IF
		END_IF
	
	//write single text line.
	3:(* Convert one PLC record to CSV format *)
		sCSVLine := '';
		fbWriter.eCmd := eEnumCmd_First;(* Write first field value *)
		IF nRow <= GVL.MAX_CSV_ROWS THEN

			FOR nColumn := 0 TO GVL.MAX_CSV_COLUMNS BY 1 DO

				sCSVField := STRING_TO_CSVFIELD( database[ nRow, nColumn ], FALSE );(* TODO: Get field value from your application *)

				(* Add new field to the record buffer *)
				fbWriter( 	pBuffer := ADR( sCSVLine ), cbBuffer := SIZEOF( sCSVLine ) - 1, putValue := sCSVField, pValue := 0, cbValue := 0,
							bCRLF := ( nColumn = GVL.MAX_CSV_COLUMNS ) );(* bCRLF == TRUE => Write CRLF after the last field value *)
				IF fbWriter.bOk THEN
					fbWriter.eCmd := eEnumCmd_Next;(* Write next field value *)
				ELSE(* Error *)
					step := 100;
					RETURN;
				END_IF

			END_FOR(* FOR nColumn := 0... *)

			(* FB_FilePuts adds allready CR (carriage return) to the written line.
			We have to replace the $R$L characters with $L character to avoid double CR. *)
			IF RIGHT( sCSVLine, 2 ) = '$R$L' THEN
				sCSVLine := REPLACE( sCSVLine, '$L', 2, LEN( sCSVLine ) - 1 );
			END_IF

			nRow := nRow + 1;(* Increment number of created records (rows) *)
			step := 4;(* Write record to the file *)

		ELSE(* All rows written => Close file *)
			step := 10;
		END_IF

	4:	(* Write single text line *)
	
		fbFilePuts( bExecute := FALSE );
		fbFilePuts( sNetId := sNetId, hFile := hFile, sLine := sCSVLine, bExecute := TRUE );
		step := 5;
	
	//waits for the line of text to finish
	5:
		fbFilePuts( bExecute := FALSE, bError => bError, nErrID => nErrID );
		IF NOT fbFilePuts.bBusy THEN
			IF NOT fbFilePuts.bError THEN
				step := 3;(* Write next record *)
			ELSE(* Error *)
				step := 100;
			END_IF
		END_IF
		
	10:
		fbFileClose( bExecute := FALSE );
		fbFileClose( sNetId := sNetId, hFile := hFile, bExecute := TRUE );
		step := 11;
	
	11:(* Wait until close not busy *)
		fbFileClose( bExecute := FALSE, bError => bError, nErrID => nErrID );
		IF ( NOT fbFileClose.bBusy ) THEN
			hFile := 0;
			step := 100;
		END_IF
		
	100: (* Error or ready step => cleanup *)
		bDone:=TRUE;
		IF ( hFile <> 0 ) THEN
			step := 10; (* Close the source file *)
		ELSE
			bBusy := FALSE;
			step := 0;	(* Ready *)
		END_IF
END_CASE
END_METHOD

METHOD reset : BOOL
VAR_INPUT
END_VAR
bDone:=FALSE;
bValidPath:=FALSE;
bWrite:=FALSE;
bError:=FALSE;
nErrId:=0;
bInProgress:=FALSE;
END_METHOD

METHOD update_database : BOOL
VAR_INPUT
	 
	user : STRING := 'N/A';
	numOfCoil : INT :=0;
	lengthOCoil : LREAL :=0;
	userNote : STRING;
	
	
END_VAR
VAR
	times: STRING(255);
	timeend: STRING(255);
END_VAR

times:=WORD_TO_STRING(startTime.wYear);
timeS:=CONCAT(times,'/');
timeS:=CONCAT(times,WORD_TO_STRING(startTime.wMonth));
timeS:=CONCAT(times,'/');
timeS:=CONCAT(times,WORD_TO_STRING(startTime.wDay));
timeS:=CONCAT(times,'/');
timeS:=CONCAT(times,WORD_TO_STRING(startTime.wHour));
timeS:=CONCAT(times,'/');
timeS:=CONCAT(times,WORD_TO_STRING(startTime.wMinute));
timeS:=CONCAT(times,'/');
timeS:=CONCAT(times,WORD_TO_STRING(startTime.wSecond));

timeend:=WORD_TO_STRING(endtime.wYear);
timeend:=CONCAT(timeend,'/');
timeend:=CONCAT(timeend,WORD_TO_STRING(endtime.wMonth));
timeend:=CONCAT(timeend,'/');
timeend:=CONCAT(timeend,WORD_TO_STRING(endtime.wDay));
timeend:=CONCAT(timeend,'/');
timeend:=CONCAT(timeend,WORD_TO_STRING(endtime.wHour));
timeend:=CONCAT(timeend,'/');
timeend:=CONCAT(timeend,WORD_TO_STRING(endtime.wMinute));
timeend:=CONCAT(timeend,'/');
timeend:=CONCAT(timeend,WORD_TO_STRING(endtime.wSecond));



database[ 0, 1 ]:=user; //user ID 
database[ 1, 1 ]:=times;
database[ 2, 1 ]:=timeend;
database[ 3, 1 ]:=WSTRING_TO_STRING(TIME_TO_WSTRING(SYSTEMTIME_TO_DT(endTime) - SYSTEMTIME_TO_DT(startTime)));
database[ 4, 1 ]:=INT_TO_STRING(numOfCoil);
database[ 5, 1 ]:=LREAL_TO_STRING(lengthOCoil);
database[ 6, 1 ]:=userNote;
END_METHOD

END_FUNCTION_BLOCK

// ---- POUs/FB_Axis.TcPOU
FUNCTION_BLOCK FB_Axis

VAR_INPUT

    //========================================================AXIS SHAPE========================================================
    coilShapeID           : INT := 0;                 // defines shape of coil attached to axis.
    pancake               : pancake_params_0;         // ID 0
    racetrack             : racetrack_params_1;       // ID 1

    //========================================================AXIS DIMENSIONS========================================================
    outerRadiusCurrent    : LREAL :=gvl.MIN_MOUNT_RADIUS/1000; // outer radius of coil

    //========================================================AXIS TAPE========================================================
    tape_info             : POINTER TO ARRAY[0..10] OF tape_info;// array of tape information
    tapeType              : INT;                      // type of tape

    //========================================================MASS========================================================
    emptyMassKG           : LREAL := 20;              // mass of the empty axis in KG
    momentInertia         : LREAL := 0;               // moment of inertia

    //========================================================AXIS CONTROL BOOL========================================================
    // sets which FB's should be executed cyclically
    powerEnable           : BOOL;                     // power enable
    resetEnable           : BOOL;                     // reset enable
    velocityEnable        : BOOL;                     // velocity enable
    haltEnable            : BOOL;                     // halt enable
    homeEnable            : BOOL;                     // home enable
    stopEnable            : BOOL;                     // stop enable
    torqueEnable          : BOOL;                     // torque enable
    posEnable             : BOOL;                     // position enable
    modmoveEnable         : BOOL;                     // move modulo enable
    test                  : BOOL;                     // test enable
    enabled               : BOOL;                     // sets whether axis is enabled
	
    //========================================================AXIS CONTROL MISC OPTIONS========================================================
    // misc options for axis
    directionB            : INT := 0;                 // direction
    direction             : MC_Direction := MC_Positive_Direction; // direction of motion
    buffermode            : MC_BufferMode := MC_Aborting;           // buffer mode
    moveOptions           : ST_MoveOptions;           // move options
    homeOptions           : ST_HomingOptions;         // homing options

    ST_SetPositionOptions : ST_SetPositionOptions;    // set position options

    //========================================================AXIS CONTROL VALUES========================================================
    // TORQUE CONTROL
    torque                : LREAL;                    // torque value
    velocityLimitHigh     : LREAL;                    // high velocity limit
    velocityLimitLow      : LREAL;                    // low velocity limit

    // SECONDARY TORQUE CONTROL SETTINGS
    acceleration          : LREAL := 1800;               // acceleration value
    deceleration          : LREAL := 1800;               // deceleration value
    torqueRamp            : LREAL := 1000;            // torque ramp value

    jerk                  : LREAL := 0;               // jerk value

    // VELOCITY CONTROL
    velocity              : LREAL;                    // velocity value

    //========================================================AXIS STATUS VARS========================================================
    actualTorque          : LREAL;                    // actual torque value
    actualVelocity        : LREAL;                    // actual velocity value
    state                 : INT;                      // state value ((1=powered,2=disabled,3=in motion,4=error))
    adsError              : BOOL;                     // ADS error flag
    adsErrorID            : UDINT;                    // ADS error ID
	errorType			  : UDINT;					  // 1= ads 2= axis 0=no error
	errorID				  : UDINT;					  // error ID, axis errors take precedence over ads errors 	
    //========================================================AXIS PARAMS========================================================
    ratedCurrent          : LREAL;                    // rated current
    torqueConstant        : LREAL;                    // torque constant
    gearRatioNum          : INT;                      // gear ratio numerator
    gearRatioDen          : INT;                      // gear ratio denominator

    //========================================================AXIS CONTROL FB========================================================
    // instantiates FB's for various axis control functions
    MCPOWER               : MC_Power;                 // power control
    MCRESET               : MC_Reset;                 // reset control
    MCHOME                : MC_Home;                  // home control
    MCVELOCITY            : MC_MoveVelocity;          // move velocity control
    MCHALT                : MC_Halt;                  // halt control
    MCSTOP                : MC_Stop;                  // stop control
    MCGETVELOCITY         : MC_ReadActualVelocity;    // read actual velocity
    MCTORQUECONTROL       : MC_TorqueControl;         // torque control
    MCPOS                 : MC_SetPosition;           // set position
    MCJOG                 : MC_Jog;                   // jog control
    MCMOVEMOD             : MC_MoveModulo;            // move modulo control
	MCReadStatus		  : MC_ReadStatus;			  // reads status from motor
	MCWriteParam		  : MC_WriteParameter;
	SoEReset			  : FB_SoEReset;			
    //========================================================AXIS========================================================
    AXIS                  : Axis_REF;                 // axis reference

END_VAR

METHOD CYLIC : BOOL
VAR_INPUT
END_VAR

VAR
	homePosition: LREAL;

	
END_VAR
Axis.ReadStatus();

powerEnable:=enabled; 

MCPOWER(Axis:=Axis,
		Enable:=powerEnable,
		Enable_Positive:=powerEnable,
		Enable_Negative:=powerEnable
		);
		
MCSTOP(Axis:=Axis,
		Execute:=stopEnable,
		Deceleration:=deceleration,
		Jerk:=jerk,Options:=moveOptions);
		
MCHALT(Axis:=Axis,
		Execute:=haltEnable,
		Deceleration:=deceleration,
		Jerk:=jerk,BufferMode:=buffermode,
		Options:=moveOptions);		

	
MCTORQUECONTROL(Axis:=Axis,
				Execute:=torqueEnable,
				ContinuousUpdate:=TRUE,
				Relative:=FALSE,
				Torque:=(torque*100)/(ratedCurrent*torqueConstant),
				TorqueRamp:=torqueRamp,
				VelocityLimitHigh:=velocityLimitHigh,
				VelocityLimitLow:=velocityLimitLow);
				
MCVELOCITY(Axis:=Axis,Execute:=FALSE);

MCVELOCITY(Axis:=Axis,
			Execute:=velocityEnable,
			Acceleration:=acceleration,
			Deceleration:=deceleration,
			Jerk:=jerk,
			Direction:=direction,
			Velocity:=velocity);
			


MCGETVELOCITY(Axis:=AXIS,
			Enable:=TRUE,
			ActualVelocity=>actualVelocity);

	 
getTorque();
stateUpdate();
findinertia();
error_check_all();


errorType:=0; //error type 1 = error inside of a FB. Error type 2 = error op axis. Error type 3= error inside of axis and on axis


IF adserror THEN
	errorType:=errorType +1 ;
	errorID:=adsErrorID;
END_IF
IF axis.Status.Error THEN
	errorType:=errorType +2;
	errorID:=axis.Status.errorid;
END_IF
END_METHOD

METHOD error_check_all : BOOL
VAR_OUTPUT
	
END_VAR

IF(powerEnable) THEN
	power_error_check(Error=>adsError,errorID=>adsErrorID);

END_IF


IF(torqueEnable) THEN
	torque_error_check(Error=>adsError,errorID=>adsErrorID);
END_IF



IF(velocityenable) THEN
	velocity_error_check(Error=>adsError,errorID=>adsErrorID);
END_IF



IF(stopenable) THEN
	stop_error_check(Error=>adsError,errorID=>adsErrorID);
END_IF




IF(posenable) THEN
	setpos_error_check(Error=>adsError,errorID=>adsErrorID);
END_IF
END_METHOD

METHOD findinertia : BOOL
VAR_INPUT
END_VAR

VAR
	cableMassKG: LREAL;
END_VAR
//to do , find mass from cable.

momentInertia:=(0.5)*(emptyMassKG+cableMassKG)*EXPT(getDistToAxis(),2);
END_METHOD

METHOD getDistToAxis : LREAL
VAR_INPUT
END_VAR
//Finds distance to axis from internal dimension and turn count vars. 

//NOTE: this only works for payoff axies. 

//output units in mm. IMPORTANT

CASE coilShapeID OF
	0:
	
	CASE directionB OF
		
	0: //Finds direction if motor is being unwound
	
	getDistToAxis:=(pancake.radius - axis.NcToPlc.ModuloActTurns*tape_info^[tapeType].tape_depth)/1000; 
	
	1: //Finds direction if motor is being wound
	
	getDistToAxis:=(pancake.radius + axis.NcToPlc.ModuloActTurns*tape_info^[tapeType].tape_depth)/1000;
	
	
	END_CASE

END_CASE
END_METHOD

METHOD getTorque : BOOL
VAR_INPUT
END_VAR
actualTorque:=(AXIS.NcToPlc.ActTorque/100)*ratedCurrent*torqueConstant;
//actualTorque:=AXIS.NcToPlc.ActTorque;
END_METHOD

METHOD halt_error_check : BOOL
VAR_INPUT
END_VAR

VAR_OUTPUT
	Error: BOOL;
	errorID: UDINT;
END_VAR
MCHALT(Axis:=Axis,Error=>Error,ErrorID=>errorID);
END_METHOD

METHOD INIT : BOOL
VAR_INPUT
END_VAR

VAR
	i: INT;
END_VAR
powerEnable:=TRUE;

//set options
ST_SetPositionOptions.ClearPositionLag:=TRUE;  

//reset axis to clear any errors
MCRESET(Axis:=AXIS,Execute:=TRUE);
MCRESET(Axis:=AXIS,Execute:=FALSE);
END_METHOD

METHOD power_error_check : BOOL
VAR_OUTPUT
	error :BOOL;
	errorID : UDINT;
END_VAR
MCPOWER(Axis:=Axis,Error=>Error,ErrorID=>errorID);
END_METHOD

METHOD reset : BOOL
VAR_INPUT
END_VAR
MCRESET(Axis:=AXIS,EXECUTE:=FALSE);
MCRESET(Axis:=AXIS,EXECUTE:=TRUE);

errorID:=0;
errorType:=0;
END_METHOD

METHOD setClear : BOOL
VAR_INPUT
END_VAR
velocityEnable:=FALSE;
stopEnable:=FALSE;
haltEnable:=FALSE;
homeEnable:= FALSE;
torqueEnable:= FALSE;
posEnable:=FALSE;
modmoveEnable:=FALSE;
END_METHOD

METHOD setFree : BOOL
VAR_INPUT
END_VAR
velocityEnable:=FALSE;
stopEnable:=FALSE;
haltEnable:=FALSE;
homeEnable:= FALSE;
torqueEnable:= FALSE;
posEnable:=FALSE;
END_METHOD

METHOD setHalt : BOOL
VAR_INPUT
END_VAR
velocityEnable:=FALSE;
stopEnable:=FALSE;
haltEnable:=TRUE;
homeEnable:= FALSE;
torqueEnable:= FALSE;
posEnable:=FALSE;
END_METHOD

METHOD setHome : BOOL
VAR_INPUT
END_VAR
velocityEnable:=FALSE;
stopEnable:=FALSE;
haltEnable:=FALSE;
homeEnable:= TRUE;
torqueEnable:= FALSE;
posEnable:=FALSE;
END_METHOD

METHOD setPos : BOOL
VAR_INPUT
	
END_VAR

VAR
	
	Done: BOOL;
	i: INT;
	busy: BOOL;
END_VAR
END_METHOD

METHOD setpos_error_check : BOOL
VAR_INPUT
END_VAR


